Axis_01_Function_Blocks ();
Axis_01_Logic ();
Axis_02_Function_Blocks ();
Axis_02_Logic ();
Axis_03_Function_Blocks ();
Axis_03_Logic ();
Axis_04_Function_Blocks ();
Axis_04_Logic ();
Axis_05_Function_Blocks ();
Axis_05_Logic ();
Axis_06_Function_Blocks ();
Axis_06_Logic ();
Axis_07_Function_Blocks ();
Axis_07_Logic ();
Axis_08_Function_Blocks ();
Axis_08_Logic ();
Axis_09_Function_Blocks ();
Axis_09_Logic ();
Axis_10_Function_Blocks ();
Axis_10_Logic ();
Axis_11_Function_Blocks ();
Axis_11_Logic ();
Axis_12_Function_Blocks ();
Axis_12_Logic ();
Axis_13_Function_Blocks ();
Axis_13_Logic ();
Axis_14_Function_Blocks ();
Axis_14_Logic ();
Axis_15_Function_Blocks ();
Axis_15_Logic ();
Axis_16_Function_Blocks ();
Axis_16_Logic ();
Group_01_Function_Blocks ();
Group_01_Logic ();
Group_02_Function_Blocks ();
Group_02_Logic ();
Group_03_Function_Blocks ();
Group_03_Logic ();
Group_04_Function_Blocks ();
Group_04_Logic ();
Group_05_Function_Blocks ();
Group_05_Logic ();
Group_06_Function_Blocks ();
Group_06_Logic ();
Group_07_Function_Blocks ();
Group_07_Logic ();
Group_08_Function_Blocks ();
Group_08_Logic ();
Indicators ();

END_PROGRAM

// ---- POUs/Axis_01_Function_Blocks.TcPOU
PROGRAM Axis_01_Function_Blocks
VAR
END_VAR

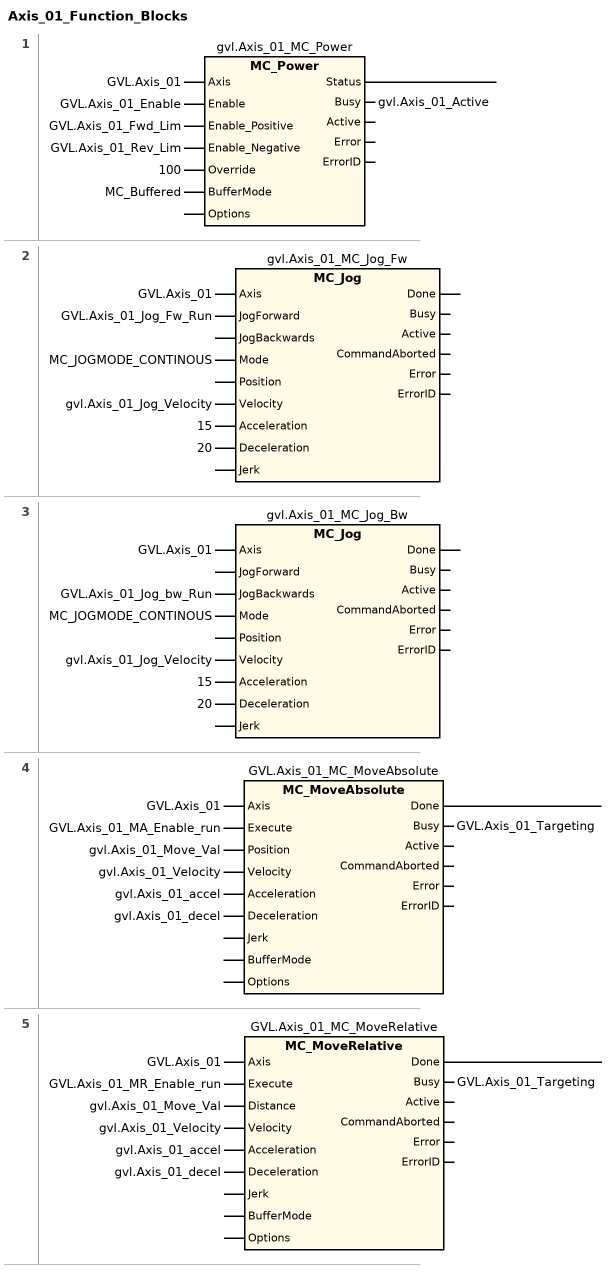
// NETWORK 1
gvl.Axis_01_MC_Power(
    Axis := GVL.Axis_01,
    Enable := GVL.Axis_01_Enable,
    Enable_Positive := GVL.Axis_01_Fwd_Lim,
    Enable_Negative := GVL.Axis_01_Rev_Lim,
    Override := 100,
    BufferMode := MC_Buffered,
    Busy => gvl.Axis_01_Active); // MC_Power

// NETWORK 2
gvl.Axis_01_MC_Jog_Fw(
    Axis := GVL.Axis_01,
    JogForward := GVL.Axis_01_Jog_Fw_Run,
    Mode := MC_JOGMODE_CONTINOUS,
    Velocity := gvl.Axis_01_Jog_Velocity,
    Acceleration := 15,
    Deceleration := 20); // MC_Jog

// NETWORK 3
gvl.Axis_01_MC_Jog_Bw(
    Axis := GVL.Axis_01,
    JogBackwards := GVL.Axis_01_Jog_bw_Run,
    Mode := MC_JOGMODE_CONTINOUS,
    Velocity := gvl.Axis_01_Jog_Velocity,
    Acceleration := 15,
    Deceleration := 20); // MC_Jog

// NETWORK 4
GVL.Axis_01_MC_MoveAbsolute(
    Axis := GVL.Axis_01,
    Execute := GVL.Axis_01_MA_Enable_run,
    Position := gvl.Axis_01_Move_Val,
    Velocity := gvl.Axis_01_Velocity,
    Acceleration := gvl.Axis_01_accel,
    Deceleration := gvl.Axis_01_decel,
    Busy => GVL.Axis_01_Targeting); // MC_MoveAbsolute

// NETWORK 5
GVL.Axis_01_MC_MoveRelative(
    Axis := GVL.Axis_01,
    Execute := GVL.Axis_01_MR_Enable_run,
    Distance := gvl.Axis_01_Move_Val,
    Velocity := gvl.Axis_01_Velocity,
    Acceleration := gvl.Axis_01_accel,
    Deceleration := gvl.Axis_01_decel,
    Busy => GVL.Axis_01_Targeting); // MC_MoveRelative

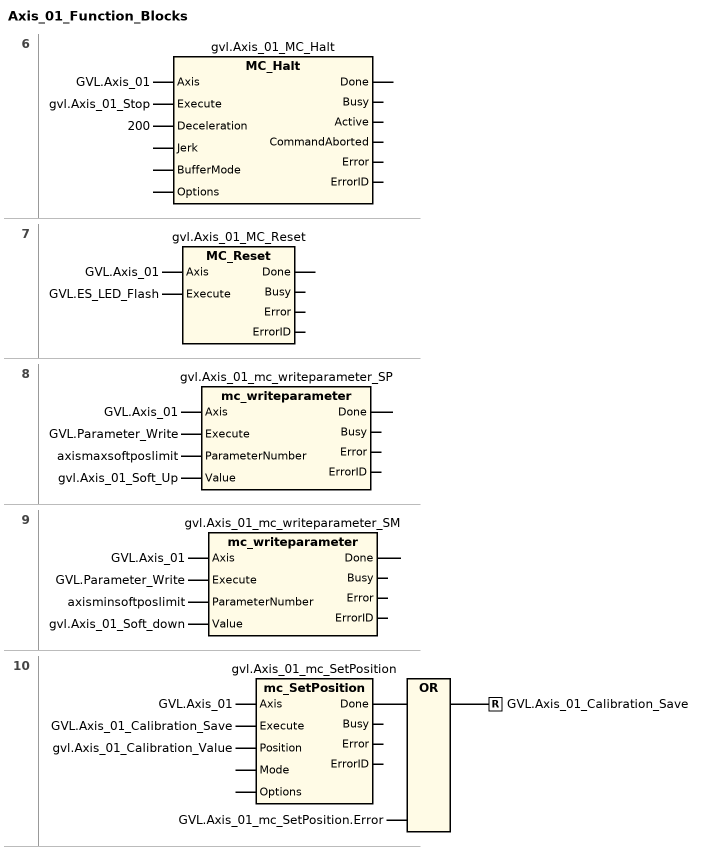
// NETWORK 6
gvl.Axis_01_MC_Halt(Axis := GVL.Axis_01, Execute := gvl.Axis_01_Stop, Deceleration := 200); // MC_Halt

// NETWORK 7
gvl.Axis_01_MC_Reset(Axis := GVL.Axis_01, Execute := GVL.ES_LED_Flash); // MC_Reset

// NETWORK 8
gvl.Axis_01_mc_writeparameter_SP(
    Axis := GVL.Axis_01,
    Execute := GVL.Parameter_Write,
    ParameterNumber := axismaxsoftposlimit,
    Value := gvl.Axis_01_Soft_Up); // mc_writeparameter

// NETWORK 9
gvl.Axis_01_mc_writeparameter_SM(
    Axis := GVL.Axis_01,
    Execute := GVL.Parameter_Write,
    ParameterNumber := axisminsoftposlimit,
    Value := gvl.Axis_01_Soft_down); // mc_writeparameter

// NETWORK 10
gvl.Axis_01_mc_SetPosition(
    Axis := GVL.Axis_01,
    Execute := GVL.Axis_01_Calibration_Save,
    Position := gvl.Axis_01_Calibration_Value); // mc_SetPosition
GVL.Axis_01_Calibration_Save R= gvl.Axis_01_mc_SetPosition.Done OR GVL.Axis_01_mc_SetPosition.Error;

END_PROGRAM

// ---- POUs/Axis_01_Logic.TcPOU
PROGRAM Axis_01_Logic
VAR
	TON_0: TON;
	TON_1: TON;
	TON_2: TON;
	TON_3: TON;
	Axis_01_Velocity_Range: LREAL;
	Axis_01_Velocity_Scale: LREAL;
	Axis_01_Velocity_Raw: LREAL;
	Axis_01_Soft_Range: LREAL;
	Axis_01_Soft_Position: LREAL;
	Axis_01_Soft_Position_In_Range: LREAL;
END_VAR

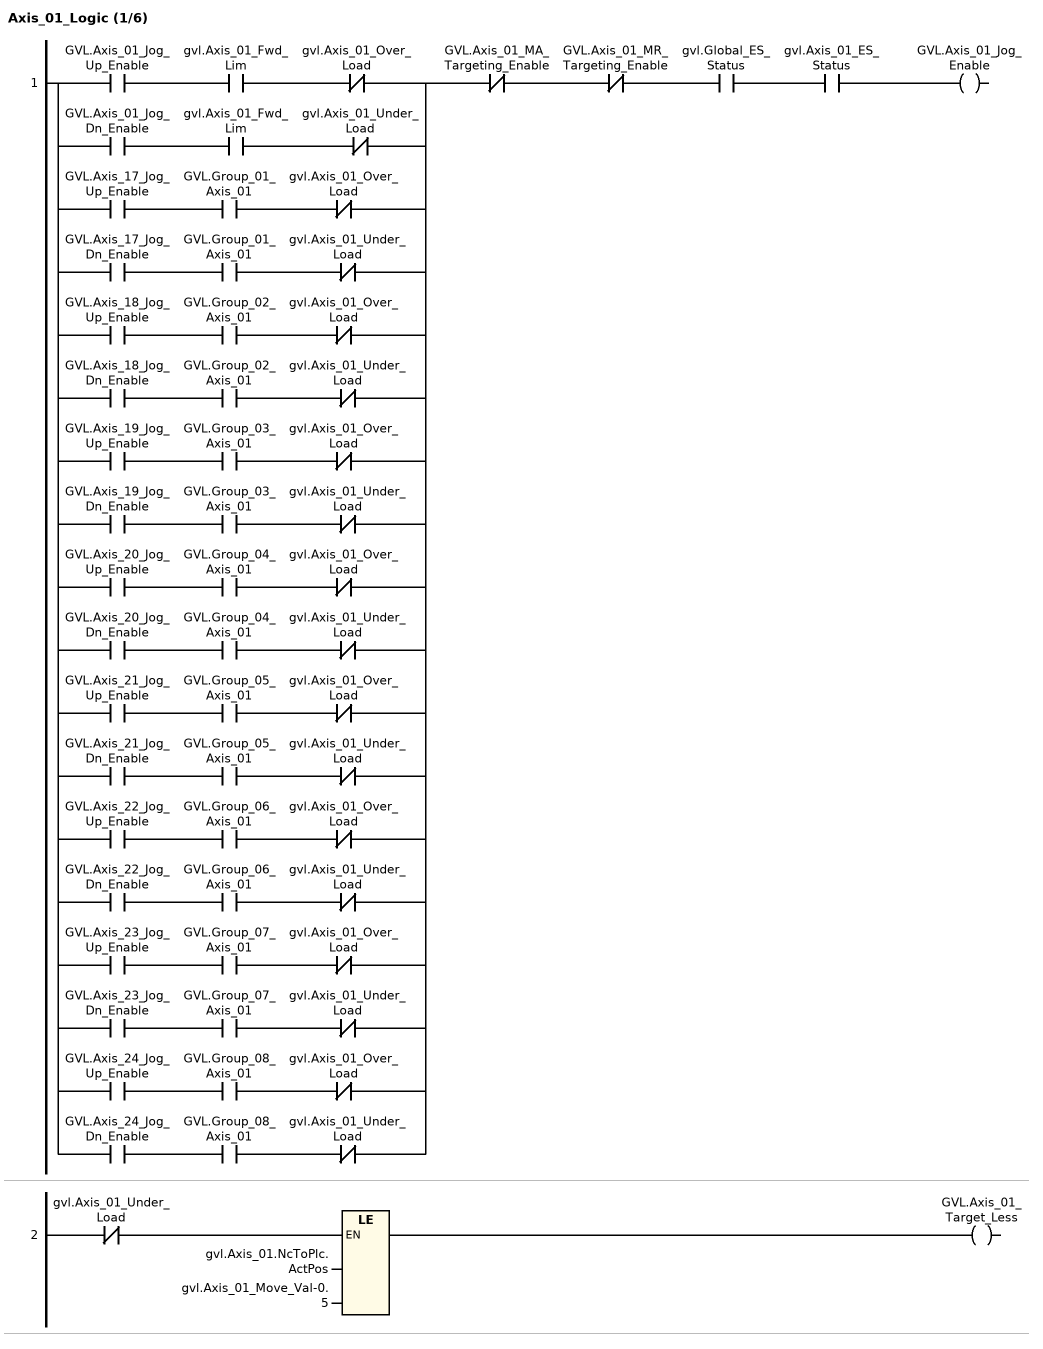
// NETWORK 1
GVL.Axis_01_Jog_Enable := (GVL.Axis_01_Jog_Up_Enable AND gvl.Axis_01_Fwd_Lim AND NOT gvl.Axis_01_Over_Load OR GVL.Axis_01_Jog_Dn_Enable AND gvl.Axis_01_Fwd_Lim AND NOT gvl.Axis_01_Under_Load OR GVL.Axis_17_Jog_Up_Enable AND GVL.Group_01_Axis_01 AND NOT gvl.Axis_01_Over_Load OR GVL.Axis_17_Jog_Dn_Enable AND GVL.Group_01_Axis_01 AND NOT gvl.Axis_01_Under_Load OR GVL.Axis_18_Jog_Up_Enable AND GVL.Group_02_Axis_01 AND NOT gvl.Axis_01_Over_Load OR GVL.Axis_18_Jog_Dn_Enable AND GVL.Group_02_Axis_01 AND NOT gvl.Axis_01_Under_Load OR GVL.Axis_19_Jog_Up_Enable AND GVL.Group_03_Axis_01 AND NOT gvl.Axis_01_Over_Load OR GVL.Axis_19_Jog_Dn_Enable AND GVL.Group_03_Axis_01 AND NOT gvl.Axis_01_Under_Load OR GVL.Axis_20_Jog_Up_Enable AND GVL.Group_04_Axis_01 AND NOT gvl.Axis_01_Over_Load OR GVL.Axis_20_Jog_Dn_Enable AND GVL.Group_04_Axis_01 AND NOT gvl.Axis_01_Under_Load OR GVL.Axis_21_Jog_Up_Enable AND GVL.Group_05_Axis_01 AND NOT gvl.Axis_01_Over_Load OR GVL.Axis_21_Jog_Dn_Enable AND GVL.Group_05_Axis_01 AND NOT gvl.Axis_01_Under_Load OR GVL.Axis_22_Jog_Up_Enable AND GVL.Group_06_Axis_01 AND NOT gvl.Axis_01_Over_Load OR GVL.Axis_22_Jog_Dn_Enable AND GVL.Group_06_Axis_01 AND NOT gvl.Axis_01_Under_Load OR GVL.Axis_23_Jog_Up_Enable AND GVL.Group_07_Axis_01 AND NOT gvl.Axis_01_Over_Load OR GVL.Axis_23_Jog_Dn_Enable AND GVL.Group_07_Axis_01 AND NOT gvl.Axis_01_Under_Load OR GVL.Axis_24_Jog_Up_Enable AND GVL.Group_08_Axis_01 AND NOT gvl.Axis_01_Over_Load OR GVL.Axis_24_Jog_Dn_Enable AND GVL.Group_08_Axis_01 AND NOT gvl.Axis_01_Under_Load) AND NOT GVL.Axis_01_MA_Targeting_Enable AND NOT GVL.Axis_01_MR_Targeting_Enable AND gvl.Global_ES_Status AND gvl.Axis_01_ES_Status;

// NETWORK 2
GVL.Axis_01_Target_Less := NOT gvl.Axis_01_Under_Load AND gvl.Axis_01.NcToPlc.ActPos <= (gvl.Axis_01_Move_Val-0.5);

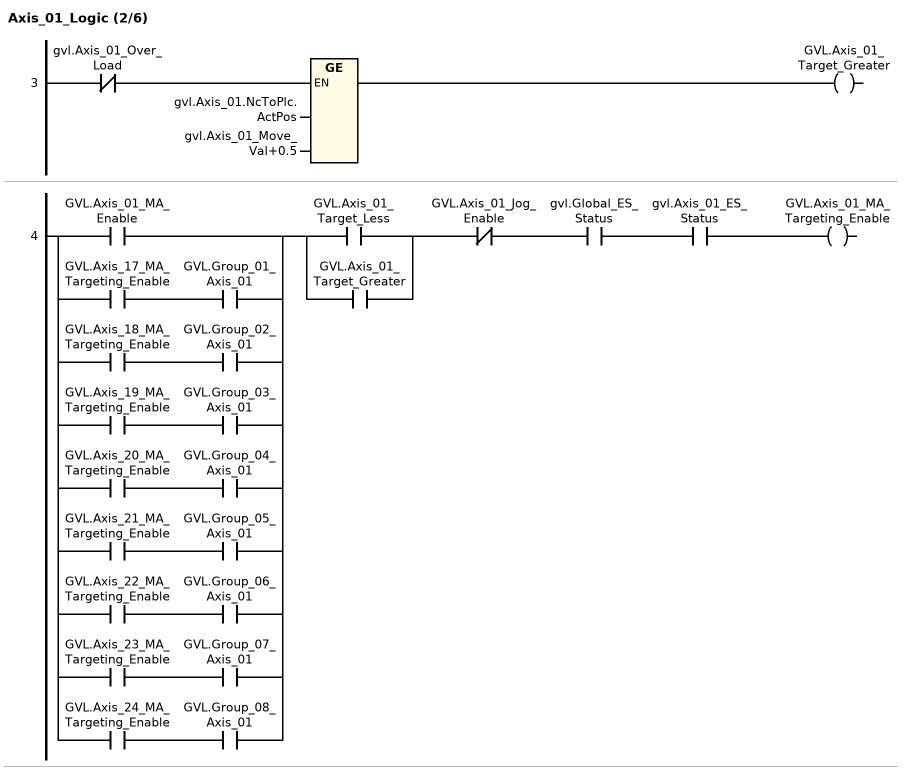
// NETWORK 3
GVL.Axis_01_Target_Greater := NOT gvl.Axis_01_Over_Load AND gvl.Axis_01.NcToPlc.ActPos >= (gvl.Axis_01_Move_Val+0.5);

// NETWORK 4
GVL.Axis_01_MA_Targeting_Enable := (GVL.Axis_01_MA_Enable OR GVL.Axis_17_MA_Targeting_Enable AND GVL.Group_01_Axis_01 OR GVL.Axis_18_MA_Targeting_Enable AND GVL.Group_02_Axis_01 OR GVL.Axis_19_MA_Targeting_Enable AND GVL.Group_03_Axis_01 OR GVL.Axis_20_MA_Targeting_Enable AND GVL.Group_04_Axis_01 OR GVL.Axis_21_MA_Targeting_Enable AND GVL.Group_05_Axis_01 OR GVL.Axis_22_MA_Targeting_Enable AND GVL.Group_06_Axis_01 OR GVL.Axis_23_MA_Targeting_Enable AND GVL.Group_07_Axis_01 OR GVL.Axis_24_MA_Targeting_Enable AND GVL.Group_08_Axis_01) AND (GVL.Axis_01_Target_Less OR GVL.Axis_01_Target_Greater) AND NOT GVL.Axis_01_Jog_Enable AND gvl.Global_ES_Status AND gvl.Axis_01_ES_Status;

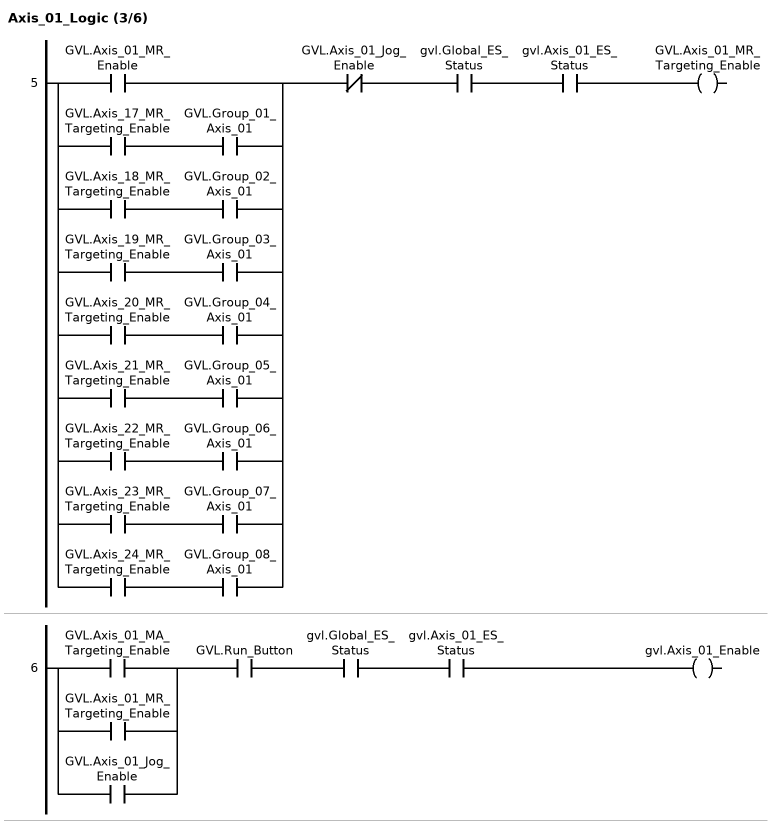
// NETWORK 5
GVL.Axis_01_MR_Targeting_Enable := (GVL.Axis_01_MR_Enable OR GVL.Axis_17_MR_Targeting_Enable AND GVL.Group_01_Axis_01 OR GVL.Axis_18_MR_Targeting_Enable AND GVL.Group_02_Axis_01 OR GVL.Axis_19_MR_Targeting_Enable AND GVL.Group_03_Axis_01 OR GVL.Axis_20_MR_Targeting_Enable AND GVL.Group_04_Axis_01 OR GVL.Axis_21_MR_Targeting_Enable AND GVL.Group_05_Axis_01 OR GVL.Axis_22_MR_Targeting_Enable AND GVL.Group_06_Axis_01 OR GVL.Axis_23_MR_Targeting_Enable AND GVL.Group_07_Axis_01 OR GVL.Axis_24_MR_Targeting_Enable AND GVL.Group_08_Axis_01) AND NOT GVL.Axis_01_Jog_Enable AND gvl.Global_ES_Status AND gvl.Axis_01_ES_Status;

// NETWORK 6
gvl.Axis_01_Enable := (GVL.Axis_01_MA_Targeting_Enable OR GVL.Axis_01_MR_Targeting_Enable OR GVL.Axis_01_Jog_Enable) AND GVL.Run_Button AND gvl.Global_ES_Status AND gvl.Axis_01_ES_Status;

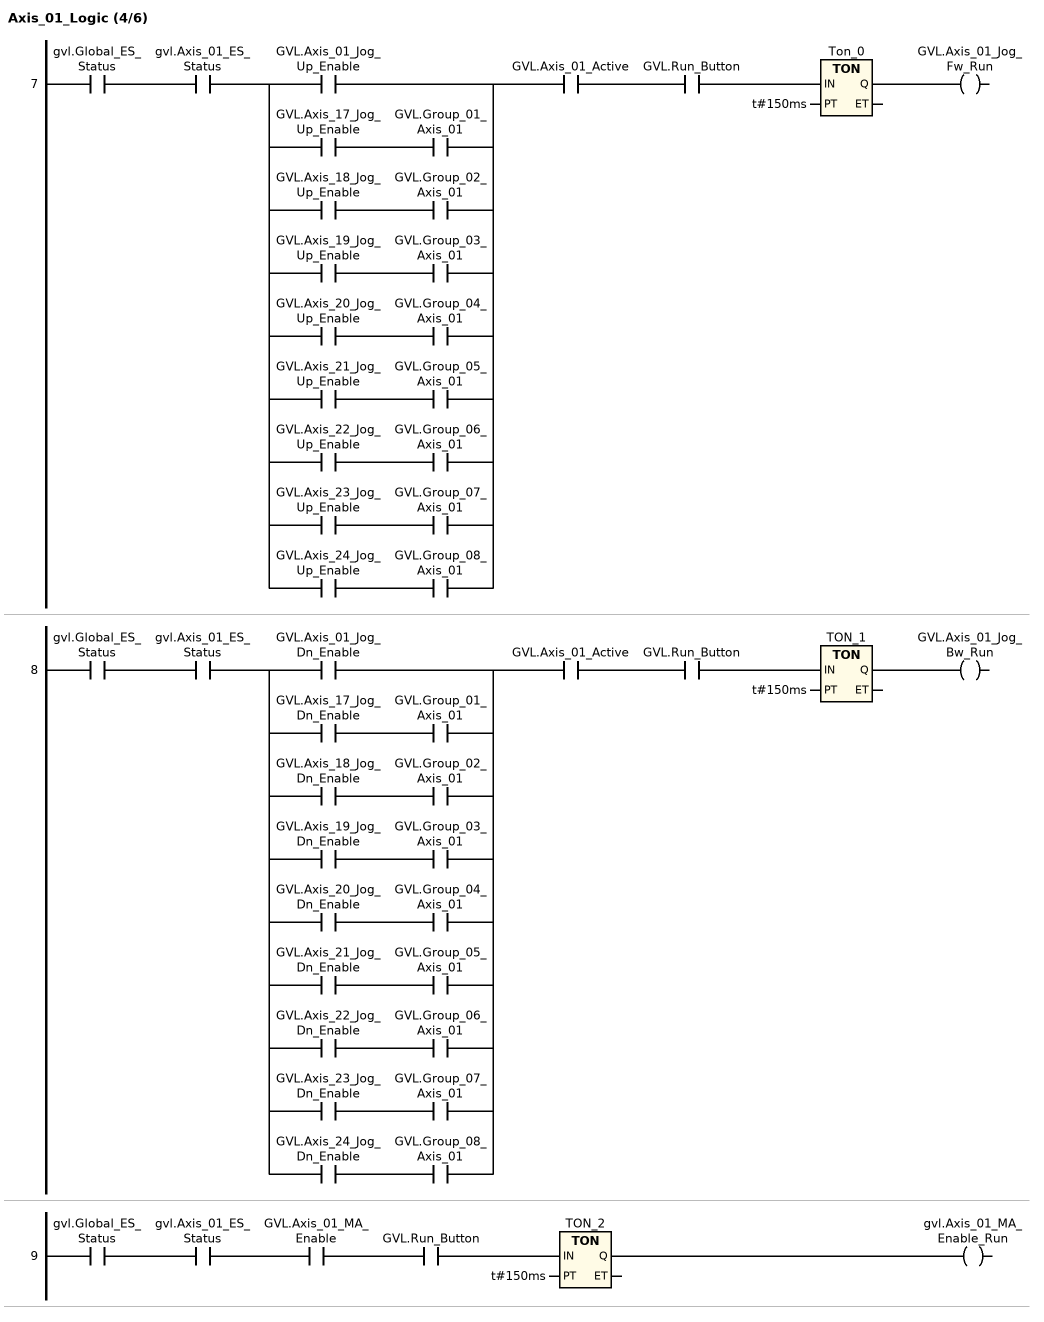
// NETWORK 7
Ton_0(IN := gvl.Global_ES_Status AND gvl.Axis_01_ES_Status AND (GVL.Axis_01_Jog_Up_Enable OR GVL.Axis_17_Jog_Up_Enable AND GVL.Group_01_Axis_01 OR GVL.Axis_18_Jog_Up_Enable AND GVL.Group_02_Axis_01 OR GVL.Axis_19_Jog_Up_Enable AND GVL.Group_03_Axis_01 OR GVL.Axis_20_Jog_Up_Enable AND GVL.Group_04_Axis_01 OR GVL.Axis_21_Jog_Up_Enable AND GVL.Group_05_Axis_01 OR GVL.Axis_22_Jog_Up_Enable AND GVL.Group_06_Axis_01 OR GVL.Axis_23_Jog_Up_Enable AND GVL.Group_07_Axis_01 OR GVL.Axis_24_Jog_Up_Enable AND GVL.Group_08_Axis_01) AND GVL.Axis_01_Active AND GVL.Run_Button, PT := t#150ms); // TON
GVL.Axis_01_Jog_Fw_Run := Ton_0.Q;

// NETWORK 8
TON_1(IN := gvl.Global_ES_Status AND gvl.Axis_01_ES_Status AND (GVL.Axis_01_Jog_Dn_Enable OR GVL.Axis_17_Jog_Dn_Enable AND GVL.Group_01_Axis_01 OR GVL.Axis_18_Jog_Dn_Enable AND GVL.Group_02_Axis_01 OR GVL.Axis_19_Jog_Dn_Enable AND GVL.Group_03_Axis_01 OR GVL.Axis_20_Jog_Dn_Enable AND GVL.Group_04_Axis_01 OR GVL.Axis_21_Jog_Dn_Enable AND GVL.Group_05_Axis_01 OR GVL.Axis_22_Jog_Dn_Enable AND GVL.Group_06_Axis_01 OR GVL.Axis_23_Jog_Dn_Enable AND GVL.Group_07_Axis_01 OR GVL.Axis_24_Jog_Dn_Enable AND GVL.Group_08_Axis_01) AND GVL.Axis_01_Active AND GVL.Run_Button, PT := t#150ms); // TON
GVL.Axis_01_Jog_Bw_Run := TON_1.Q;

// NETWORK 9
TON_2(IN := gvl.Global_ES_Status AND gvl.Axis_01_ES_Status AND GVL.Axis_01_MA_Enable AND GVL.Run_Button, PT := t#150ms); // TON
gvl.Axis_01_MA_Enable_Run := TON_2.Q;

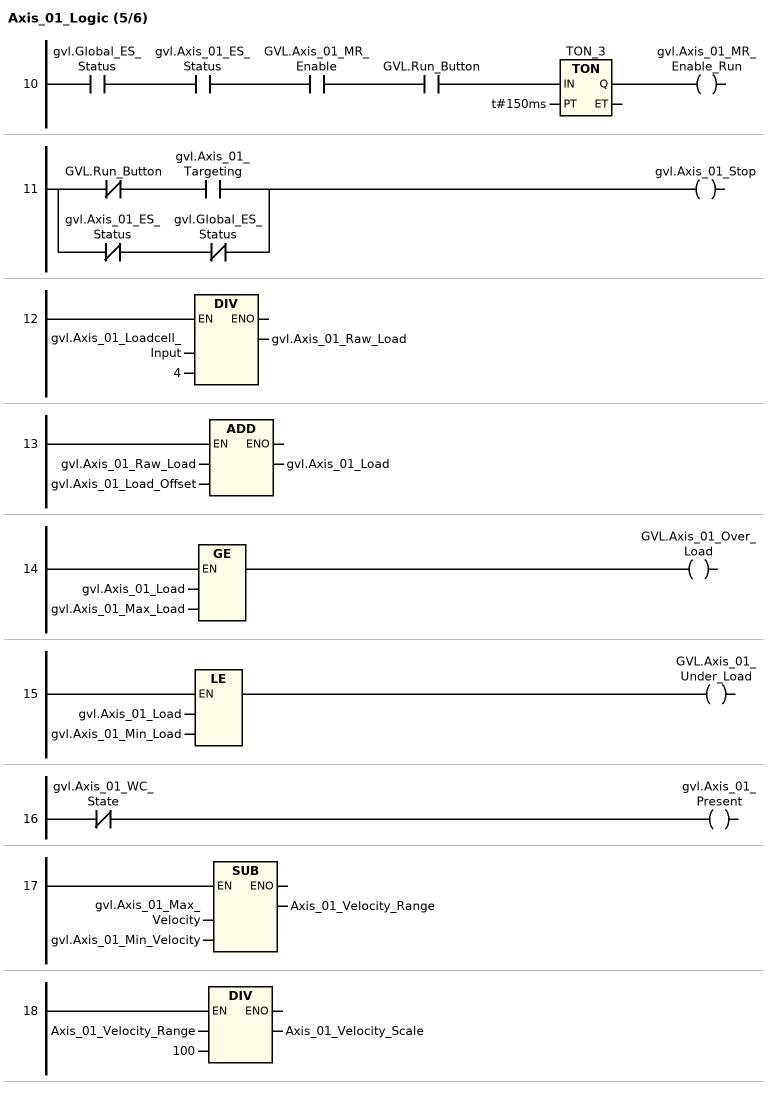
// NETWORK 10
TON_3(IN := gvl.Global_ES_Status AND gvl.Axis_01_ES_Status AND GVL.Axis_01_MR_Enable AND GVL.Run_Button, PT := t#150ms); // TON
gvl.Axis_01_MR_Enable_Run := TON_3.Q;

// NETWORK 11
gvl.Axis_01_Stop := NOT GVL.Run_Button AND gvl.Axis_01_Targeting OR NOT gvl.Axis_01_ES_Status AND NOT gvl.Global_ES_Status;

// NETWORK 12
gvl.Axis_01_Raw_Load := gvl.Axis_01_Loadcell_Input / 4;

// NETWORK 13
gvl.Axis_01_Load := gvl.Axis_01_Raw_Load + gvl.Axis_01_Load_Offset;

// NETWORK 14
GVL.Axis_01_Over_Load := gvl.Axis_01_Load >= gvl.Axis_01_Max_Load;

// NETWORK 15
GVL.Axis_01_Under_Load := gvl.Axis_01_Load <= gvl.Axis_01_Min_Load;

// NETWORK 16
gvl.Axis_01_Present := NOT gvl.Axis_01_WC_State;

// NETWORK 17
Axis_01_Velocity_Range := gvl.Axis_01_Max_Velocity - gvl.Axis_01_Min_Velocity;

// NETWORK 18
Axis_01_Velocity_Scale := Axis_01_Velocity_Range / 100;

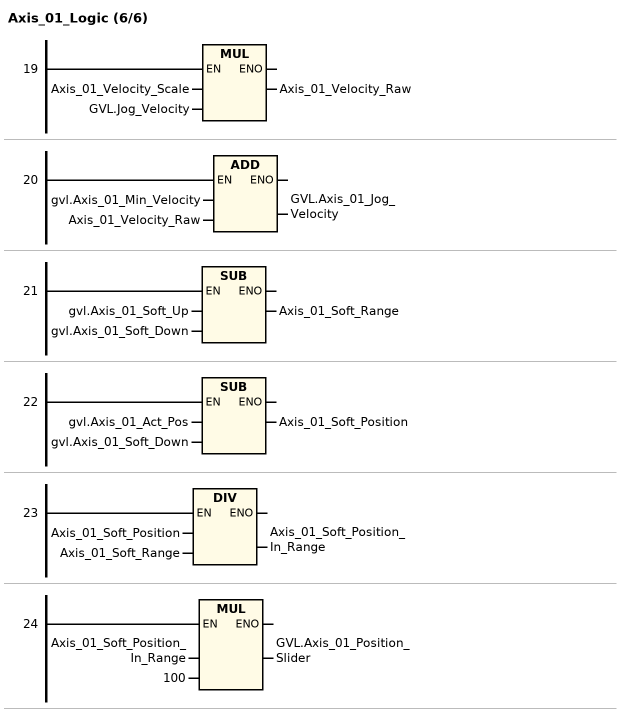
// NETWORK 19
Axis_01_Velocity_Raw := Axis_01_Velocity_Scale * GVL.Jog_Velocity;

// NETWORK 20
GVL.Axis_01_Jog_Velocity := gvl.Axis_01_Min_Velocity + Axis_01_Velocity_Raw;

// NETWORK 21
Axis_01_Soft_Range := gvl.Axis_01_Soft_Up - gvl.Axis_01_Soft_Down;

// NETWORK 22
Axis_01_Soft_Position := gvl.Axis_01_Act_Pos - gvl.Axis_01_Soft_Down;

// NETWORK 23
Axis_01_Soft_Position_In_Range := Axis_01_Soft_Position / Axis_01_Soft_Range;

// NETWORK 24
GVL.Axis_01_Position_Slider := Axis_01_Soft_Position_In_Range * 100;

END_PROGRAM

// ---- POUs/Axis_02_Function_Blocks.TcPOU
PROGRAM Axis_02_Function_Blocks
VAR
END_VAR

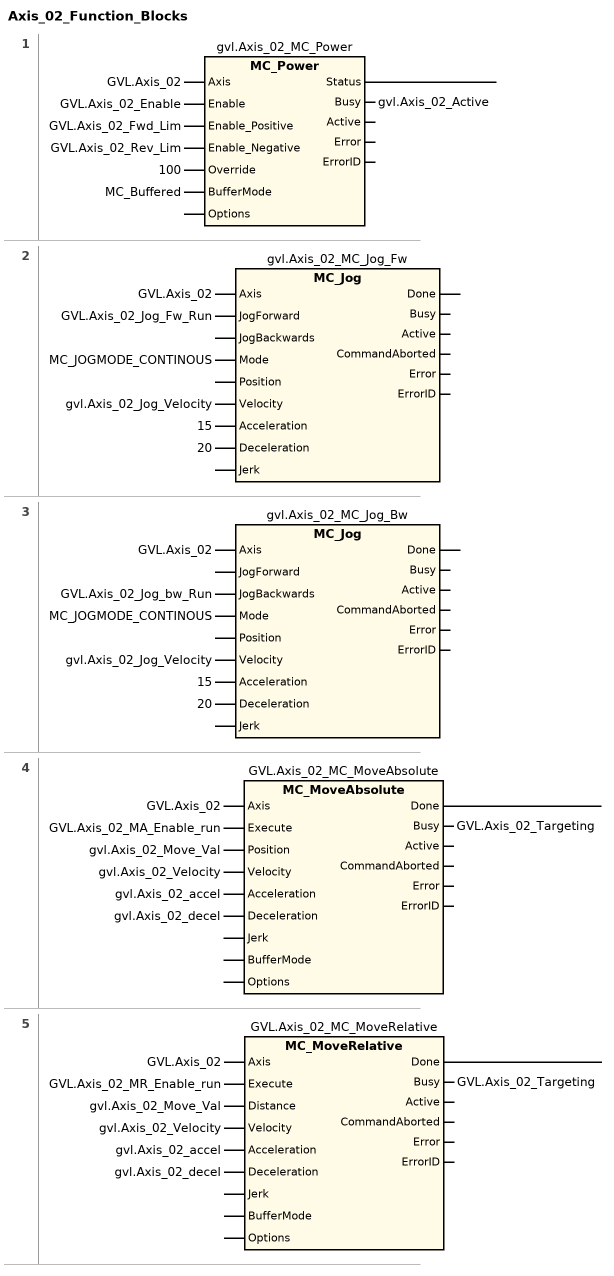
// NETWORK 1
gvl.Axis_02_MC_Power(
    Axis := GVL.Axis_02,
    Enable := GVL.Axis_02_Enable,
    Enable_Positive := GVL.Axis_02_Fwd_Lim,
    Enable_Negative := GVL.Axis_02_Rev_Lim,
    Override := 100,
    BufferMode := MC_Buffered,
    Busy => gvl.Axis_02_Active); // MC_Power

// NETWORK 2
gvl.Axis_02_MC_Jog_Fw(
    Axis := GVL.Axis_02,
    JogForward := GVL.Axis_02_Jog_Fw_Run,
    Mode := MC_JOGMODE_CONTINOUS,
    Velocity := gvl.Axis_02_Jog_Velocity,
    Acceleration := 15,
    Deceleration := 20); // MC_Jog

// NETWORK 3
gvl.Axis_02_MC_Jog_Bw(
    Axis := GVL.Axis_02,
    JogBackwards := GVL.Axis_02_Jog_bw_Run,
    Mode := MC_JOGMODE_CONTINOUS,
    Velocity := gvl.Axis_02_Jog_Velocity,
    Acceleration := 15,
    Deceleration := 20); // MC_Jog

// NETWORK 4
GVL.Axis_02_MC_MoveAbsolute(
    Axis := GVL.Axis_02,
    Execute := GVL.Axis_02_MA_Enable_run,
    Position := gvl.Axis_02_Move_Val,
    Velocity := gvl.Axis_02_Velocity,
    Acceleration := gvl.Axis_02_accel,
    Deceleration := gvl.Axis_02_decel,
    Busy => GVL.Axis_02_Targeting); // MC_MoveAbsolute

// NETWORK 5
GVL.Axis_02_MC_MoveRelative(
    Axis := GVL.Axis_02,
    Execute := GVL.Axis_02_MR_Enable_run,
    Distance := gvl.Axis_02_Move_Val,
    Velocity := gvl.Axis_02_Velocity,
    Acceleration := gvl.Axis_02_accel,
    Deceleration := gvl.Axis_02_decel,
    Busy => GVL.Axis_02_Targeting); // MC_MoveRelative

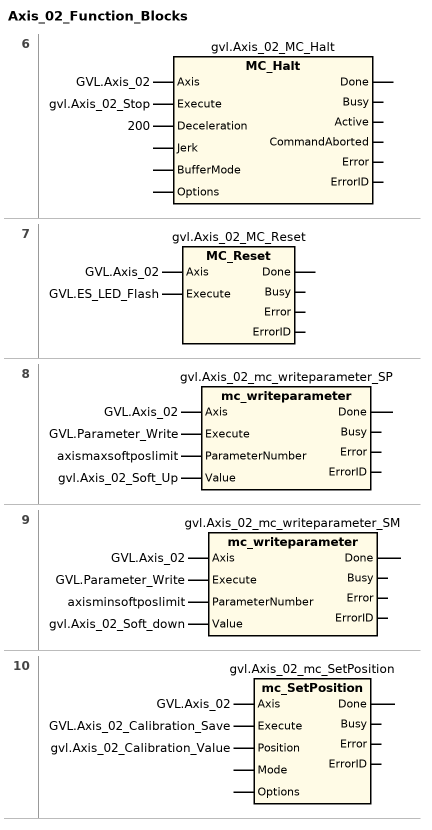
// NETWORK 6
gvl.Axis_02_MC_Halt(Axis := GVL.Axis_02, Execute := gvl.Axis_02_Stop, Deceleration := 200); // MC_Halt

// NETWORK 7
gvl.Axis_02_MC_Reset(Axis := GVL.Axis_02, Execute := GVL.ES_LED_Flash); // MC_Reset

// NETWORK 8
gvl.Axis_02_mc_writeparameter_SP(
    Axis := GVL.Axis_02,
    Execute := GVL.Parameter_Write,
    ParameterNumber := axismaxsoftposlimit,
    Value := gvl.Axis_02_Soft_Up); // mc_writeparameter

// NETWORK 9
gvl.Axis_02_mc_writeparameter_SM(
    Axis := GVL.Axis_02,
    Execute := GVL.Parameter_Write,
    ParameterNumber := axisminsoftposlimit,
    Value := gvl.Axis_02_Soft_down); // mc_writeparameter

// NETWORK 10
gvl.Axis_02_mc_SetPosition(
    Axis := GVL.Axis_02,
    Execute := GVL.Axis_02_Calibration_Save,
    Position := gvl.Axis_02_Calibration_Value); // mc_SetPosition

END_PROGRAM

// ---- POUs/Axis_02_Logic.TcPOU
PROGRAM Axis_02_Logic
VAR
	TON_0: TON;
	TON_1: TON;
	TON_2: TON;
	TON_3: TON;
	Axis_02_Velocity_Range: LREAL;
	Axis_02_Velocity_Scale: LREAL;
	Axis_02_Velocity_Raw: LREAL;
	Axis_02_Soft_Range: LREAL;
	Axis_02_Soft_Position: LREAL;
	Axis_02_Soft_Position_In_Range: LREAL;
END_VAR

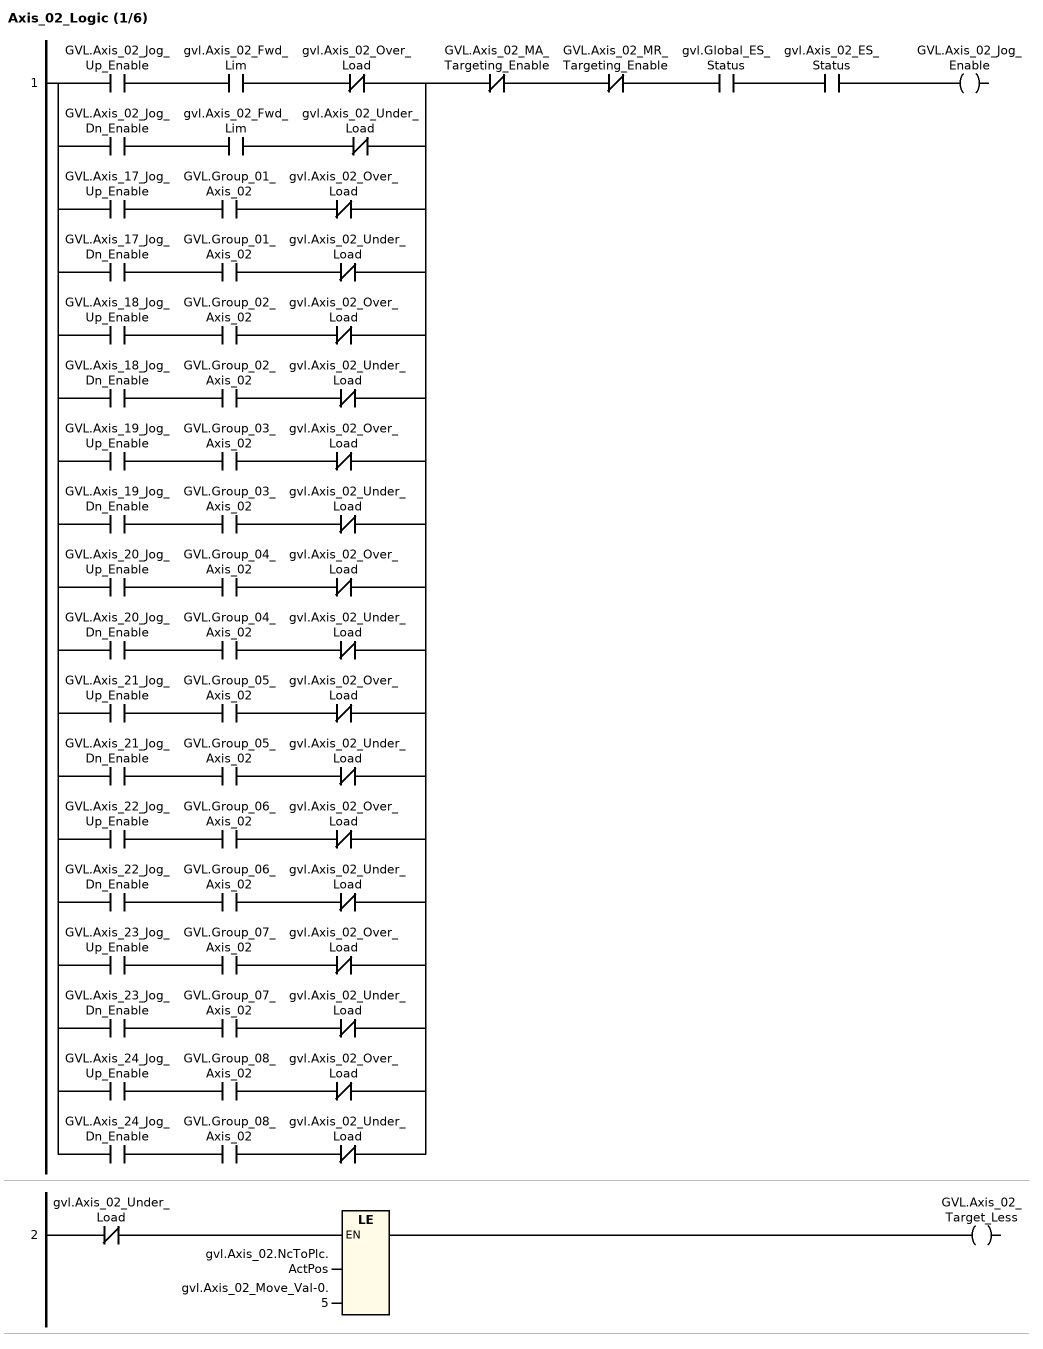
// NETWORK 1
GVL.Axis_02_Jog_Enable := (GVL.Axis_02_Jog_Up_Enable AND gvl.Axis_02_Fwd_Lim AND NOT gvl.Axis_02_Over_Load OR GVL.Axis_02_Jog_Dn_Enable AND gvl.Axis_02_Fwd_Lim AND NOT gvl.Axis_02_Under_Load OR GVL.Axis_17_Jog_Up_Enable AND GVL.Group_01_Axis_02 AND NOT gvl.Axis_02_Over_Load OR GVL.Axis_17_Jog_Dn_Enable AND GVL.Group_01_Axis_02 AND NOT gvl.Axis_02_Under_Load OR GVL.Axis_18_Jog_Up_Enable AND GVL.Group_02_Axis_02 AND NOT gvl.Axis_02_Over_Load OR GVL.Axis_18_Jog_Dn_Enable AND GVL.Group_02_Axis_02 AND NOT gvl.Axis_02_Under_Load OR GVL.Axis_19_Jog_Up_Enable AND GVL.Group_03_Axis_02 AND NOT gvl.Axis_02_Over_Load OR GVL.Axis_19_Jog_Dn_Enable AND GVL.Group_03_Axis_02 AND NOT gvl.Axis_02_Under_Load OR GVL.Axis_20_Jog_Up_Enable AND GVL.Group_04_Axis_02 AND NOT gvl.Axis_02_Over_Load OR GVL.Axis_20_Jog_Dn_Enable AND GVL.Group_04_Axis_02 AND NOT gvl.Axis_02_Under_Load OR GVL.Axis_21_Jog_Up_Enable AND GVL.Group_05_Axis_02 AND NOT gvl.Axis_02_Over_Load OR GVL.Axis_21_Jog_Dn_Enable AND GVL.Group_05_Axis_02 AND NOT gvl.Axis_02_Under_Load OR GVL.Axis_22_Jog_Up_Enable AND GVL.Group_06_Axis_02 AND NOT gvl.Axis_02_Over_Load OR GVL.Axis_22_Jog_Dn_Enable AND GVL.Group_06_Axis_02 AND NOT gvl.Axis_02_Under_Load OR GVL.Axis_23_Jog_Up_Enable AND GVL.Group_07_Axis_02 AND NOT gvl.Axis_02_Over_Load OR GVL.Axis_23_Jog_Dn_Enable AND GVL.Group_07_Axis_02 AND NOT gvl.Axis_02_Under_Load OR GVL.Axis_24_Jog_Up_Enable AND GVL.Group_08_Axis_02 AND NOT gvl.Axis_02_Over_Load OR GVL.Axis_24_Jog_Dn_Enable AND GVL.Group_08_Axis_02 AND NOT gvl.Axis_02_Under_Load) AND NOT GVL.Axis_02_MA_Targeting_Enable AND NOT GVL.Axis_02_MR_Targeting_Enable AND gvl.Global_ES_Status AND gvl.Axis_02_ES_Status;

// NETWORK 2
GVL.Axis_02_Target_Less := NOT gvl.Axis_02_Under_Load AND gvl.Axis_02.NcToPlc.ActPos <= (gvl.Axis_02_Move_Val-0.5);

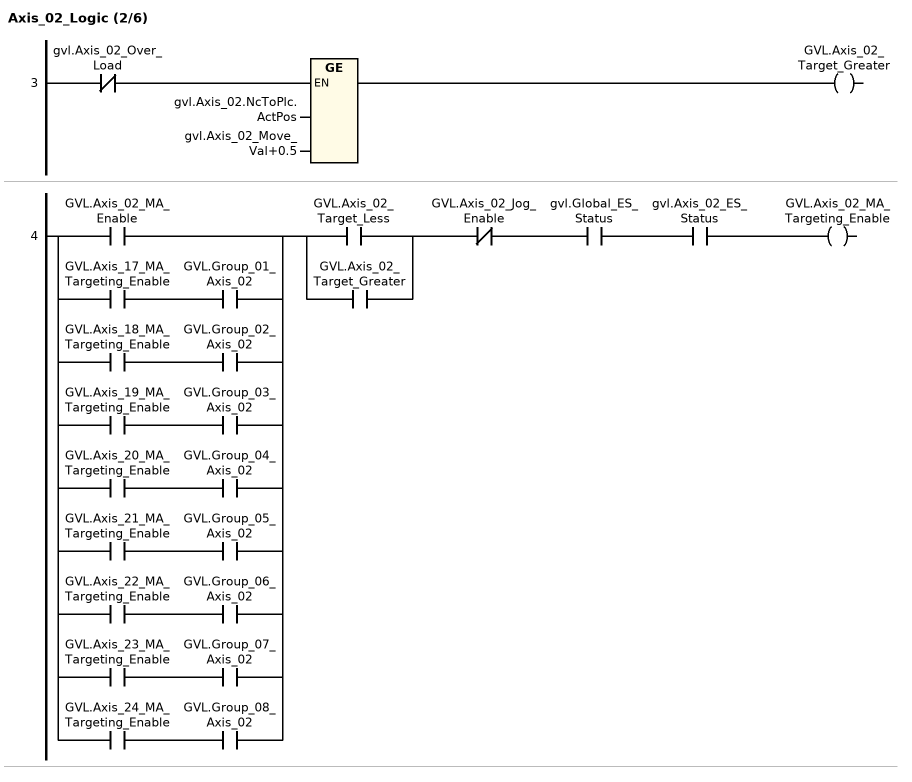
// NETWORK 3
GVL.Axis_02_Target_Greater := NOT gvl.Axis_02_Over_Load AND gvl.Axis_02.NcToPlc.ActPos >= (gvl.Axis_02_Move_Val+0.5);

// NETWORK 4
GVL.Axis_02_MA_Targeting_Enable := (GVL.Axis_02_MA_Enable OR GVL.Axis_17_MA_Targeting_Enable AND GVL.Group_01_Axis_02 OR GVL.Axis_18_MA_Targeting_Enable AND GVL.Group_02_Axis_02 OR GVL.Axis_19_MA_Targeting_Enable AND GVL.Group_03_Axis_02 OR GVL.Axis_20_MA_Targeting_Enable AND GVL.Group_04_Axis_02 OR GVL.Axis_21_MA_Targeting_Enable AND GVL.Group_05_Axis_02 OR GVL.Axis_22_MA_Targeting_Enable AND GVL.Group_06_Axis_02 OR GVL.Axis_23_MA_Targeting_Enable AND GVL.Group_07_Axis_02 OR GVL.Axis_24_MA_Targeting_Enable AND GVL.Group_08_Axis_02) AND (GVL.Axis_02_Target_Less OR GVL.Axis_02_Target_Greater) AND NOT GVL.Axis_02_Jog_Enable AND gvl.Global_ES_Status AND gvl.Axis_02_ES_Status;

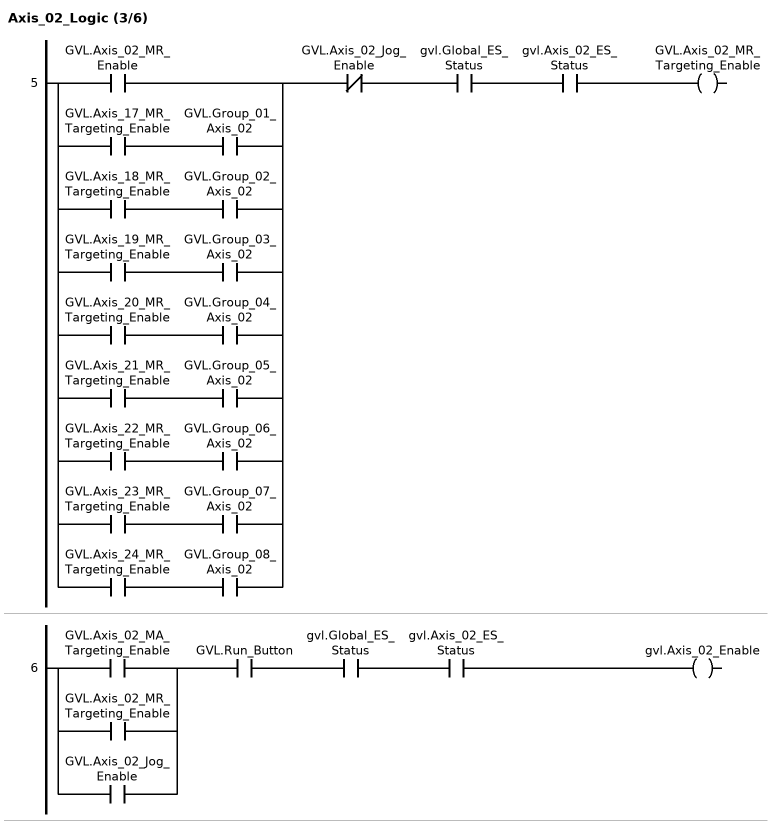
// NETWORK 5
GVL.Axis_02_MR_Targeting_Enable := (GVL.Axis_02_MR_Enable OR GVL.Axis_17_MR_Targeting_Enable AND GVL.Group_01_Axis_02 OR GVL.Axis_18_MR_Targeting_Enable AND GVL.Group_02_Axis_02 OR GVL.Axis_19_MR_Targeting_Enable AND GVL.Group_03_Axis_02 OR GVL.Axis_20_MR_Targeting_Enable AND GVL.Group_04_Axis_02 OR GVL.Axis_21_MR_Targeting_Enable AND GVL.Group_05_Axis_02 OR GVL.Axis_22_MR_Targeting_Enable AND GVL.Group_06_Axis_02 OR GVL.Axis_23_MR_Targeting_Enable AND GVL.Group_07_Axis_02 OR GVL.Axis_24_MR_Targeting_Enable AND GVL.Group_08_Axis_02) AND NOT GVL.Axis_02_Jog_Enable AND gvl.Global_ES_Status AND gvl.Axis_02_ES_Status;

// NETWORK 6
gvl.Axis_02_Enable := (GVL.Axis_02_MA_Targeting_Enable OR GVL.Axis_02_MR_Targeting_Enable OR GVL.Axis_02_Jog_Enable) AND GVL.Run_Button AND gvl.Global_ES_Status AND gvl.Axis_02_ES_Status;

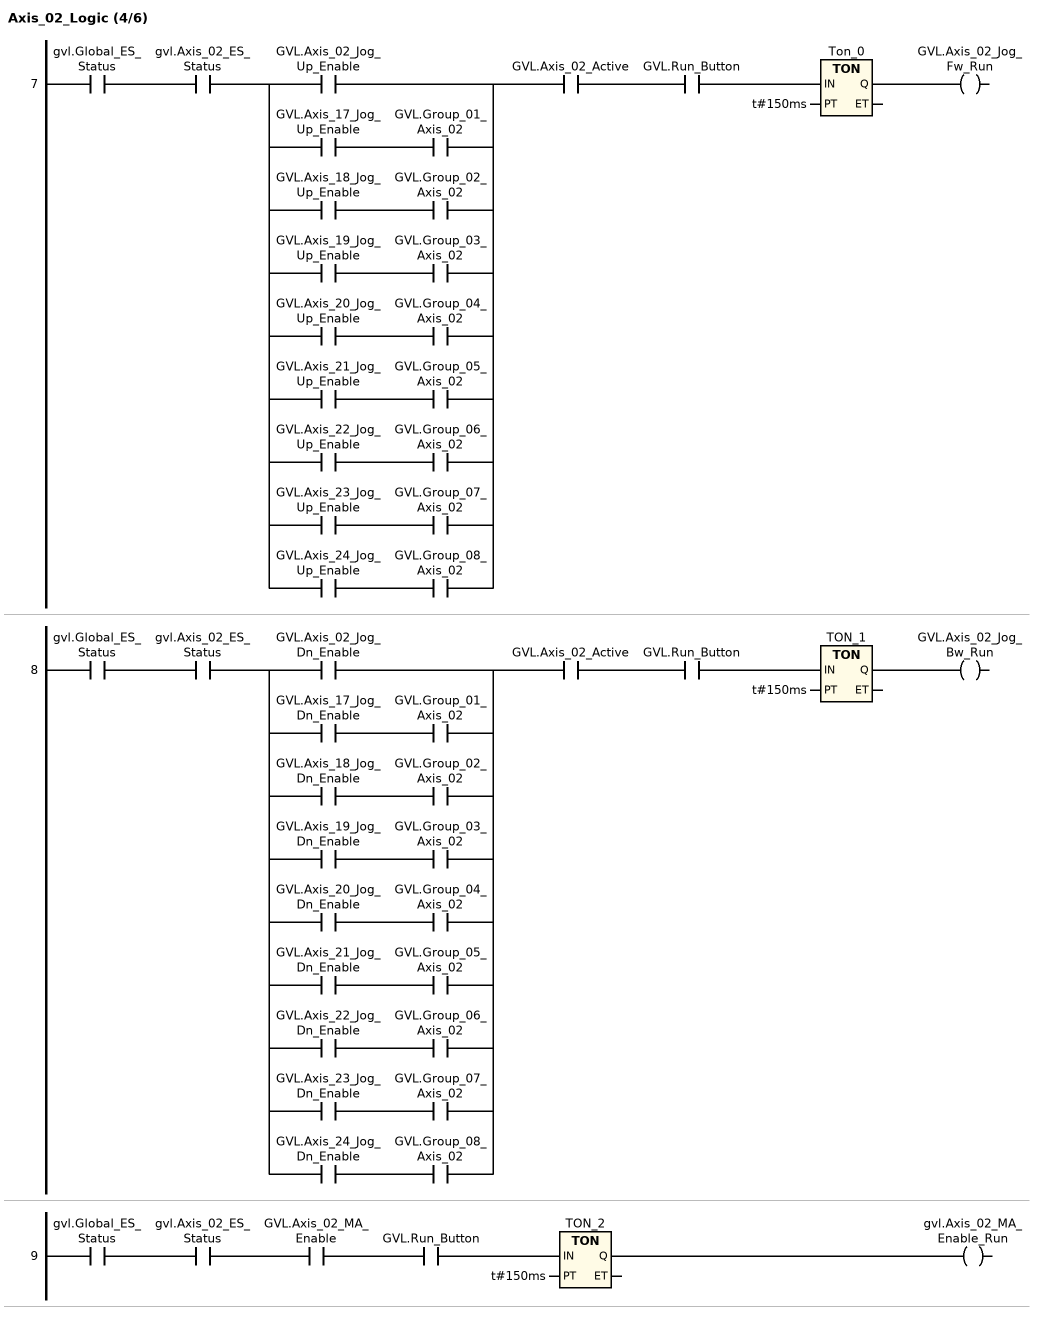
// NETWORK 7
Ton_0(IN := gvl.Global_ES_Status AND gvl.Axis_02_ES_Status AND (GVL.Axis_02_Jog_Up_Enable OR GVL.Axis_17_Jog_Up_Enable AND GVL.Group_01_Axis_02 OR GVL.Axis_18_Jog_Up_Enable AND GVL.Group_02_Axis_02 OR GVL.Axis_19_Jog_Up_Enable AND GVL.Group_03_Axis_02 OR GVL.Axis_20_Jog_Up_Enable AND GVL.Group_04_Axis_02 OR GVL.Axis_21_Jog_Up_Enable AND GVL.Group_05_Axis_02 OR GVL.Axis_22_Jog_Up_Enable AND GVL.Group_06_Axis_02 OR GVL.Axis_23_Jog_Up_Enable AND GVL.Group_07_Axis_02 OR GVL.Axis_24_Jog_Up_Enable AND GVL.Group_08_Axis_02) AND GVL.Axis_02_Active AND GVL.Run_Button, PT := t#150ms); // TON
GVL.Axis_02_Jog_Fw_Run := Ton_0.Q;

// NETWORK 8
TON_1(IN := gvl.Global_ES_Status AND gvl.Axis_02_ES_Status AND (GVL.Axis_02_Jog_Dn_Enable OR GVL.Axis_17_Jog_Dn_Enable AND GVL.Group_01_Axis_02 OR GVL.Axis_18_Jog_Dn_Enable AND GVL.Group_02_Axis_02 OR GVL.Axis_19_Jog_Dn_Enable AND GVL.Group_03_Axis_02 OR GVL.Axis_20_Jog_Dn_Enable AND GVL.Group_04_Axis_02 OR GVL.Axis_21_Jog_Dn_Enable AND GVL.Group_05_Axis_02 OR GVL.Axis_22_Jog_Dn_Enable AND GVL.Group_06_Axis_02 OR GVL.Axis_23_Jog_Dn_Enable AND GVL.Group_07_Axis_02 OR GVL.Axis_24_Jog_Dn_Enable AND GVL.Group_08_Axis_02) AND GVL.Axis_02_Active AND GVL.Run_Button, PT := t#150ms); // TON
GVL.Axis_02_Jog_Bw_Run := TON_1.Q;

// NETWORK 9
TON_2(IN := gvl.Global_ES_Status AND gvl.Axis_02_ES_Status AND GVL.Axis_02_MA_Enable AND GVL.Run_Button, PT := t#150ms); // TON
gvl.Axis_02_MA_Enable_Run := TON_2.Q;

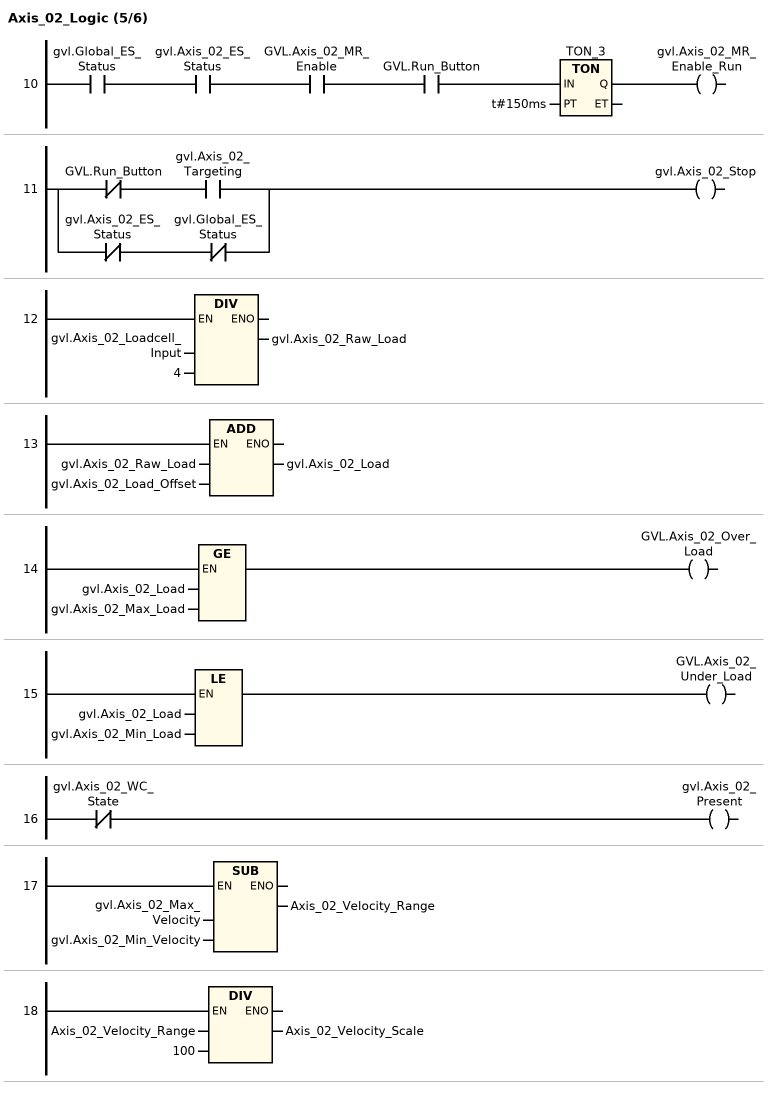
// NETWORK 10
TON_3(IN := gvl.Global_ES_Status AND gvl.Axis_02_ES_Status AND GVL.Axis_02_MR_Enable AND GVL.Run_Button, PT := t#150ms); // TON
gvl.Axis_02_MR_Enable_Run := TON_3.Q;

// NETWORK 11
gvl.Axis_02_Stop := NOT GVL.Run_Button AND gvl.Axis_02_Targeting OR NOT gvl.Axis_02_ES_Status AND NOT gvl.Global_ES_Status;

// NETWORK 12
gvl.Axis_02_Raw_Load := gvl.Axis_02_Loadcell_Input / 4;

// NETWORK 13
gvl.Axis_02_Load := gvl.Axis_02_Raw_Load + gvl.Axis_02_Load_Offset;

// NETWORK 14
GVL.Axis_02_Over_Load := gvl.Axis_02_Load >= gvl.Axis_02_Max_Load;

// NETWORK 15
GVL.Axis_02_Under_Load := gvl.Axis_02_Load <= gvl.Axis_02_Min_Load;

// NETWORK 16
gvl.Axis_02_Present := NOT gvl.Axis_02_WC_State;

// NETWORK 17
Axis_02_Velocity_Range := gvl.Axis_02_Max_Velocity - gvl.Axis_02_Min_Velocity;

// NETWORK 18
Axis_02_Velocity_Scale := Axis_02_Velocity_Range / 100;

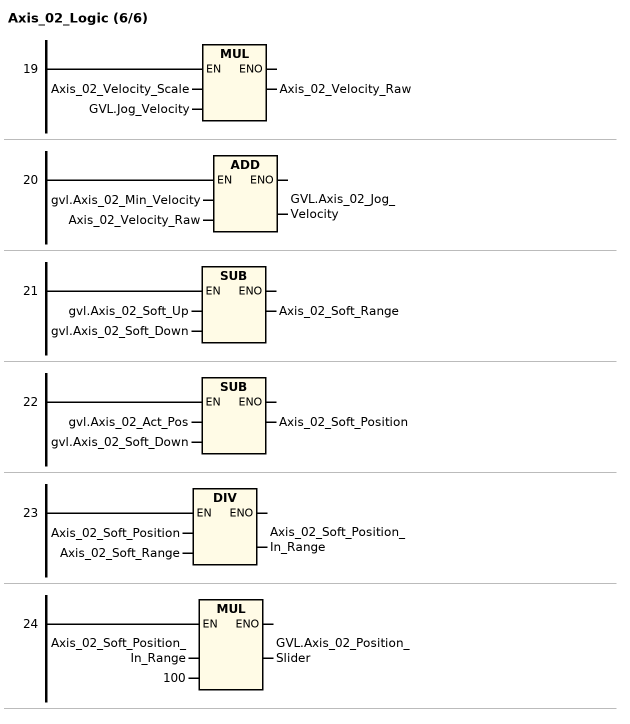
// NETWORK 19
Axis_02_Velocity_Raw := Axis_02_Velocity_Scale * GVL.Jog_Velocity;

// NETWORK 20
GVL.Axis_02_Jog_Velocity := gvl.Axis_02_Min_Velocity + Axis_02_Velocity_Raw;

// NETWORK 21
Axis_02_Soft_Range := gvl.Axis_02_Soft_Up - gvl.Axis_02_Soft_Down;

// NETWORK 22
Axis_02_Soft_Position := gvl.Axis_02_Act_Pos - gvl.Axis_02_Soft_Down;

// NETWORK 23
Axis_02_Soft_Position_In_Range := Axis_02_Soft_Position / Axis_02_Soft_Range;

// NETWORK 24
GVL.Axis_02_Position_Slider := Axis_02_Soft_Position_In_Range * 100;

END_PROGRAM

// ---- POUs/Axis_03_Function_Blocks.TcPOU
PROGRAM Axis_03_Function_Blocks
VAR
END_VAR

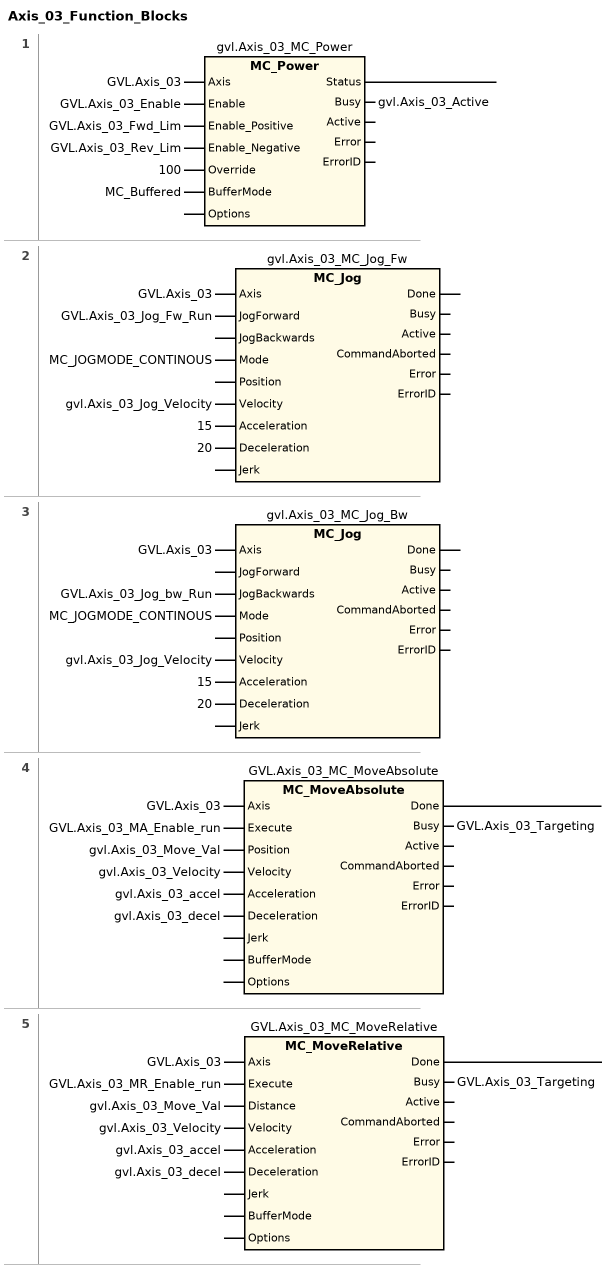
// NETWORK 1
gvl.Axis_03_MC_Power(
    Axis := GVL.Axis_03,
    Enable := GVL.Axis_03_Enable,
    Enable_Positive := GVL.Axis_03_Fwd_Lim,
    Enable_Negative := GVL.Axis_03_Rev_Lim,
    Override := 100,
    BufferMode := MC_Buffered,
    Busy => gvl.Axis_03_Active); // MC_Power

// NETWORK 2
gvl.Axis_03_MC_Jog_Fw(
    Axis := GVL.Axis_03,
    JogForward := GVL.Axis_03_Jog_Fw_Run,
    Mode := MC_JOGMODE_CONTINOUS,
    Velocity := gvl.Axis_03_Jog_Velocity,
    Acceleration := 15,
    Deceleration := 20); // MC_Jog

// NETWORK 3
gvl.Axis_03_MC_Jog_Bw(
    Axis := GVL.Axis_03,
    JogBackwards := GVL.Axis_03_Jog_bw_Run,
    Mode := MC_JOGMODE_CONTINOUS,
    Velocity := gvl.Axis_03_Jog_Velocity,
    Acceleration := 15,
    Deceleration := 20); // MC_Jog

// NETWORK 4
GVL.Axis_03_MC_MoveAbsolute(
    Axis := GVL.Axis_03,
    Execute := GVL.Axis_03_MA_Enable_run,
    Position := gvl.Axis_03_Move_Val,
    Velocity := gvl.Axis_03_Velocity,
    Acceleration := gvl.Axis_03_accel,
    Deceleration := gvl.Axis_03_decel,
    Busy => GVL.Axis_03_Targeting); // MC_MoveAbsolute

// NETWORK 5
GVL.Axis_03_MC_MoveRelative(
    Axis := GVL.Axis_03,
    Execute := GVL.Axis_03_MR_Enable_run,
    Distance := gvl.Axis_03_Move_Val,
    Velocity := gvl.Axis_03_Velocity,
    Acceleration := gvl.Axis_03_accel,
    Deceleration := gvl.Axis_03_decel,
    Busy => GVL.Axis_03_Targeting); // MC_MoveRelative

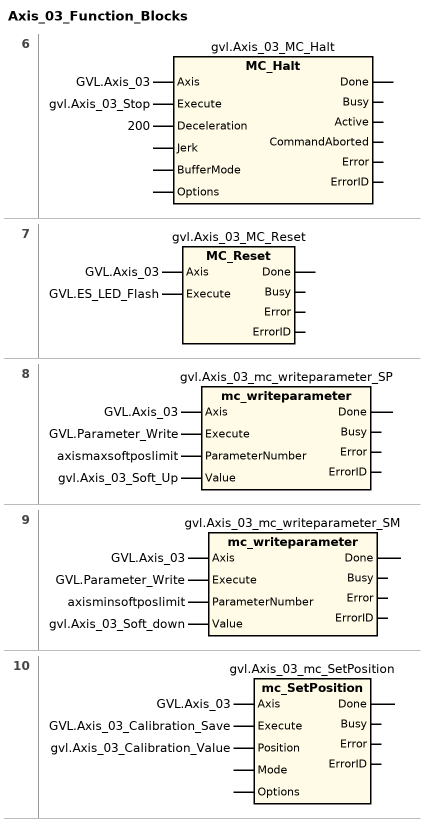
// NETWORK 6
gvl.Axis_03_MC_Halt(Axis := GVL.Axis_03, Execute := gvl.Axis_03_Stop, Deceleration := 200); // MC_Halt

// NETWORK 7
gvl.Axis_03_MC_Reset(Axis := GVL.Axis_03, Execute := GVL.ES_LED_Flash); // MC_Reset

// NETWORK 8
gvl.Axis_03_mc_writeparameter_SP(
    Axis := GVL.Axis_03,
    Execute := GVL.Parameter_Write,
    ParameterNumber := axismaxsoftposlimit,
    Value := gvl.Axis_03_Soft_Up); // mc_writeparameter

// NETWORK 9
gvl.Axis_03_mc_writeparameter_SM(
    Axis := GVL.Axis_03,
    Execute := GVL.Parameter_Write,
    ParameterNumber := axisminsoftposlimit,
    Value := gvl.Axis_03_Soft_down); // mc_writeparameter

// NETWORK 10
gvl.Axis_03_mc_SetPosition(
    Axis := GVL.Axis_03,
    Execute := GVL.Axis_03_Calibration_Save,
    Position := gvl.Axis_03_Calibration_Value); // mc_SetPosition

END_PROGRAM

// ---- POUs/Axis_03_Logic.TcPOU
PROGRAM Axis_03_Logic
VAR
	TON_0: TON;
	TON_1: TON;
	TON_2: TON;
	TON_3: TON;
	Axis_03_Velocity_Range: LREAL;
	Axis_03_Velocity_Scale: LREAL;
	Axis_03_Velocity_Raw: LREAL;
	Axis_03_Soft_Range: LREAL;
	Axis_03_Soft_Position: LREAL;
	Axis_03_Soft_Position_In_Range: LREAL;
END_VAR

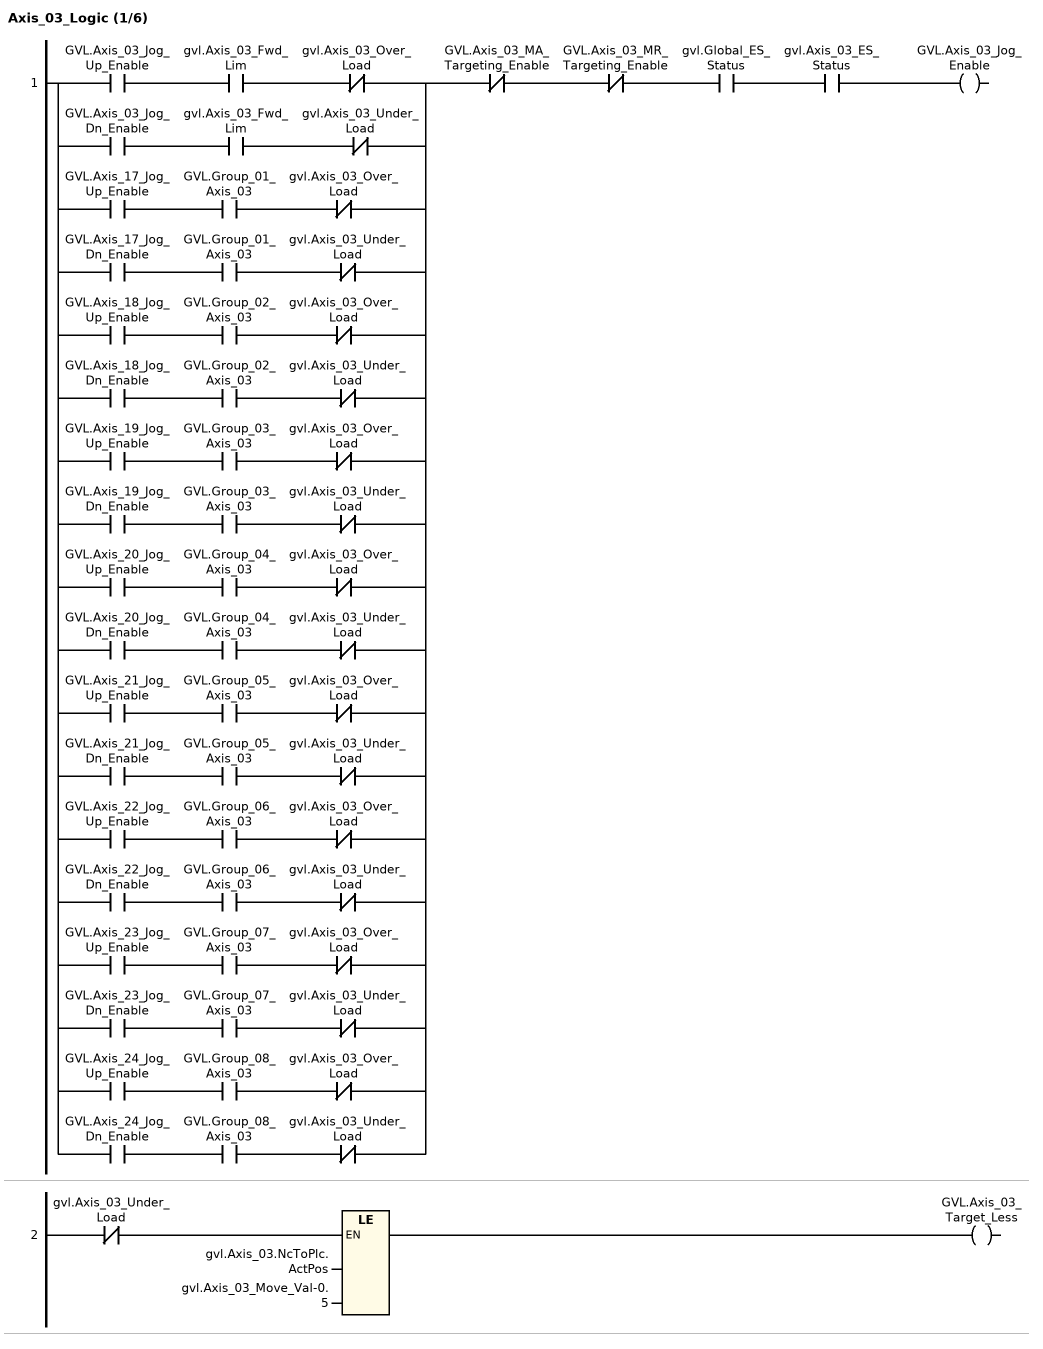
// NETWORK 1
GVL.Axis_03_Jog_Enable := (GVL.Axis_03_Jog_Up_Enable AND gvl.Axis_03_Fwd_Lim AND NOT gvl.Axis_03_Over_Load OR GVL.Axis_03_Jog_Dn_Enable AND gvl.Axis_03_Fwd_Lim AND NOT gvl.Axis_03_Under_Load OR GVL.Axis_17_Jog_Up_Enable AND GVL.Group_01_Axis_03 AND NOT gvl.Axis_03_Over_Load OR GVL.Axis_17_Jog_Dn_Enable AND GVL.Group_01_Axis_03 AND NOT gvl.Axis_03_Under_Load OR GVL.Axis_18_Jog_Up_Enable AND GVL.Group_02_Axis_03 AND NOT gvl.Axis_03_Over_Load OR GVL.Axis_18_Jog_Dn_Enable AND GVL.Group_02_Axis_03 AND NOT gvl.Axis_03_Under_Load OR GVL.Axis_19_Jog_Up_Enable AND GVL.Group_03_Axis_03 AND NOT gvl.Axis_03_Over_Load OR GVL.Axis_19_Jog_Dn_Enable AND GVL.Group_03_Axis_03 AND NOT gvl.Axis_03_Under_Load OR GVL.Axis_20_Jog_Up_Enable AND GVL.Group_04_Axis_03 AND NOT gvl.Axis_03_Over_Load OR GVL.Axis_20_Jog_Dn_Enable AND GVL.Group_04_Axis_03 AND NOT gvl.Axis_03_Under_Load OR GVL.Axis_21_Jog_Up_Enable AND GVL.Group_05_Axis_03 AND NOT gvl.Axis_03_Over_Load OR GVL.Axis_21_Jog_Dn_Enable AND GVL.Group_05_Axis_03 AND NOT gvl.Axis_03_Under_Load OR GVL.Axis_22_Jog_Up_Enable AND GVL.Group_06_Axis_03 AND NOT gvl.Axis_03_Over_Load OR GVL.Axis_22_Jog_Dn_Enable AND GVL.Group_06_Axis_03 AND NOT gvl.Axis_03_Under_Load OR GVL.Axis_23_Jog_Up_Enable AND GVL.Group_07_Axis_03 AND NOT gvl.Axis_03_Over_Load OR GVL.Axis_23_Jog_Dn_Enable AND GVL.Group_07_Axis_03 AND NOT gvl.Axis_03_Under_Load OR GVL.Axis_24_Jog_Up_Enable AND GVL.Group_08_Axis_03 AND NOT gvl.Axis_03_Over_Load OR GVL.Axis_24_Jog_Dn_Enable AND GVL.Group_08_Axis_03 AND NOT gvl.Axis_03_Under_Load) AND NOT GVL.Axis_03_MA_Targeting_Enable AND NOT GVL.Axis_03_MR_Targeting_Enable AND gvl.Global_ES_Status AND gvl.Axis_03_ES_Status;

// NETWORK 2
GVL.Axis_03_Target_Less := NOT gvl.Axis_03_Under_Load AND gvl.Axis_03.NcToPlc.ActPos <= (gvl.Axis_03_Move_Val-0.5);

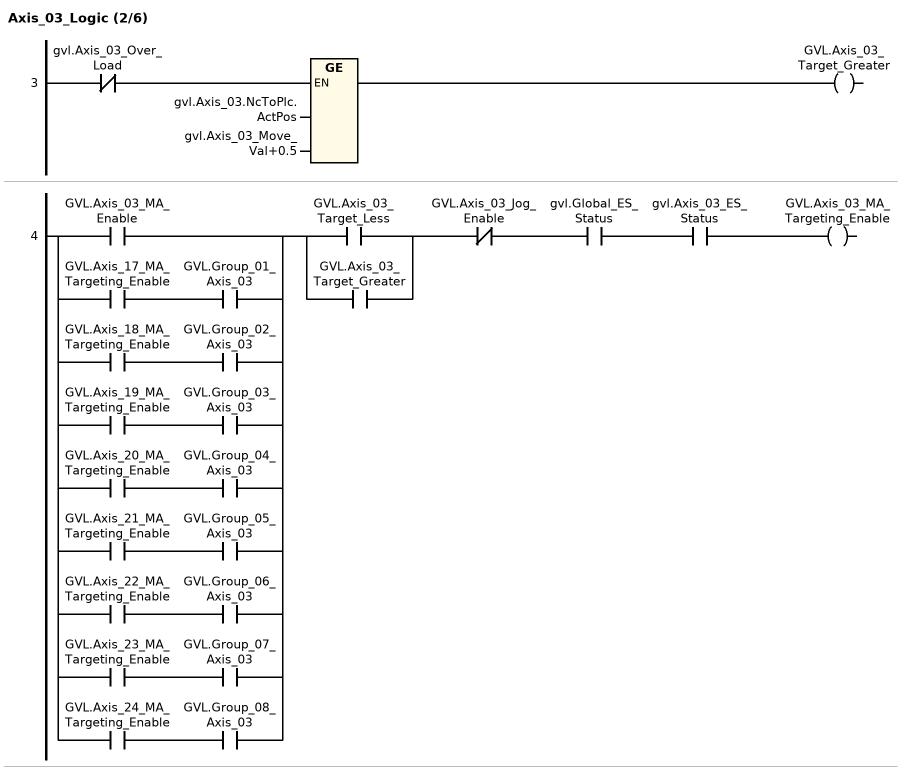
// NETWORK 3
GVL.Axis_03_Target_Greater := NOT gvl.Axis_03_Over_Load AND gvl.Axis_03.NcToPlc.ActPos >= (gvl.Axis_03_Move_Val+0.5);

// NETWORK 4
GVL.Axis_03_MA_Targeting_Enable := (GVL.Axis_03_MA_Enable OR GVL.Axis_17_MA_Targeting_Enable AND GVL.Group_01_Axis_03 OR GVL.Axis_18_MA_Targeting_Enable AND GVL.Group_02_Axis_03 OR GVL.Axis_19_MA_Targeting_Enable AND GVL.Group_03_Axis_03 OR GVL.Axis_20_MA_Targeting_Enable AND GVL.Group_04_Axis_03 OR GVL.Axis_21_MA_Targeting_Enable AND GVL.Group_05_Axis_03 OR GVL.Axis_22_MA_Targeting_Enable AND GVL.Group_06_Axis_03 OR GVL.Axis_23_MA_Targeting_Enable AND GVL.Group_07_Axis_03 OR GVL.Axis_24_MA_Targeting_Enable AND GVL.Group_08_Axis_03) AND (GVL.Axis_03_Target_Less OR GVL.Axis_03_Target_Greater) AND NOT GVL.Axis_03_Jog_Enable AND gvl.Global_ES_Status AND gvl.Axis_03_ES_Status;

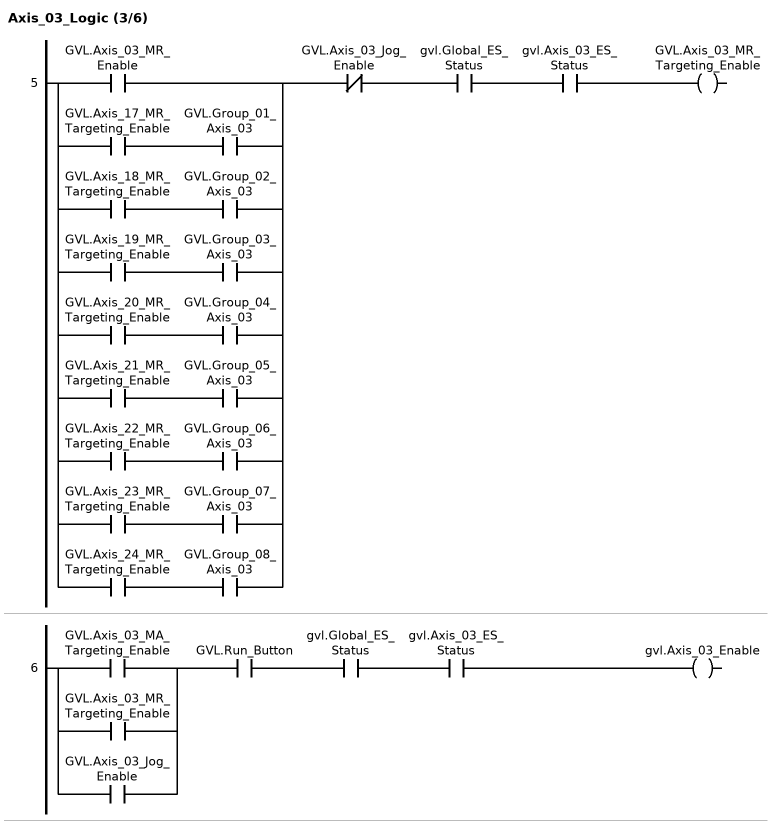
// NETWORK 5
GVL.Axis_03_MR_Targeting_Enable := (GVL.Axis_03_MR_Enable OR GVL.Axis_17_MR_Targeting_Enable AND GVL.Group_01_Axis_03 OR GVL.Axis_18_MR_Targeting_Enable AND GVL.Group_02_Axis_03 OR GVL.Axis_19_MR_Targeting_Enable AND GVL.Group_03_Axis_03 OR GVL.Axis_20_MR_Targeting_Enable AND GVL.Group_04_Axis_03 OR GVL.Axis_21_MR_Targeting_Enable AND GVL.Group_05_Axis_03 OR GVL.Axis_22_MR_Targeting_Enable AND GVL.Group_06_Axis_03 OR GVL.Axis_23_MR_Targeting_Enable AND GVL.Group_07_Axis_03 OR GVL.Axis_24_MR_Targeting_Enable AND GVL.Group_08_Axis_03) AND NOT GVL.Axis_03_Jog_Enable AND gvl.Global_ES_Status AND gvl.Axis_03_ES_Status;

// NETWORK 6
gvl.Axis_03_Enable := (GVL.Axis_03_MA_Targeting_Enable OR GVL.Axis_03_MR_Targeting_Enable OR GVL.Axis_03_Jog_Enable) AND GVL.Run_Button AND gvl.Global_ES_Status AND gvl.Axis_03_ES_Status;

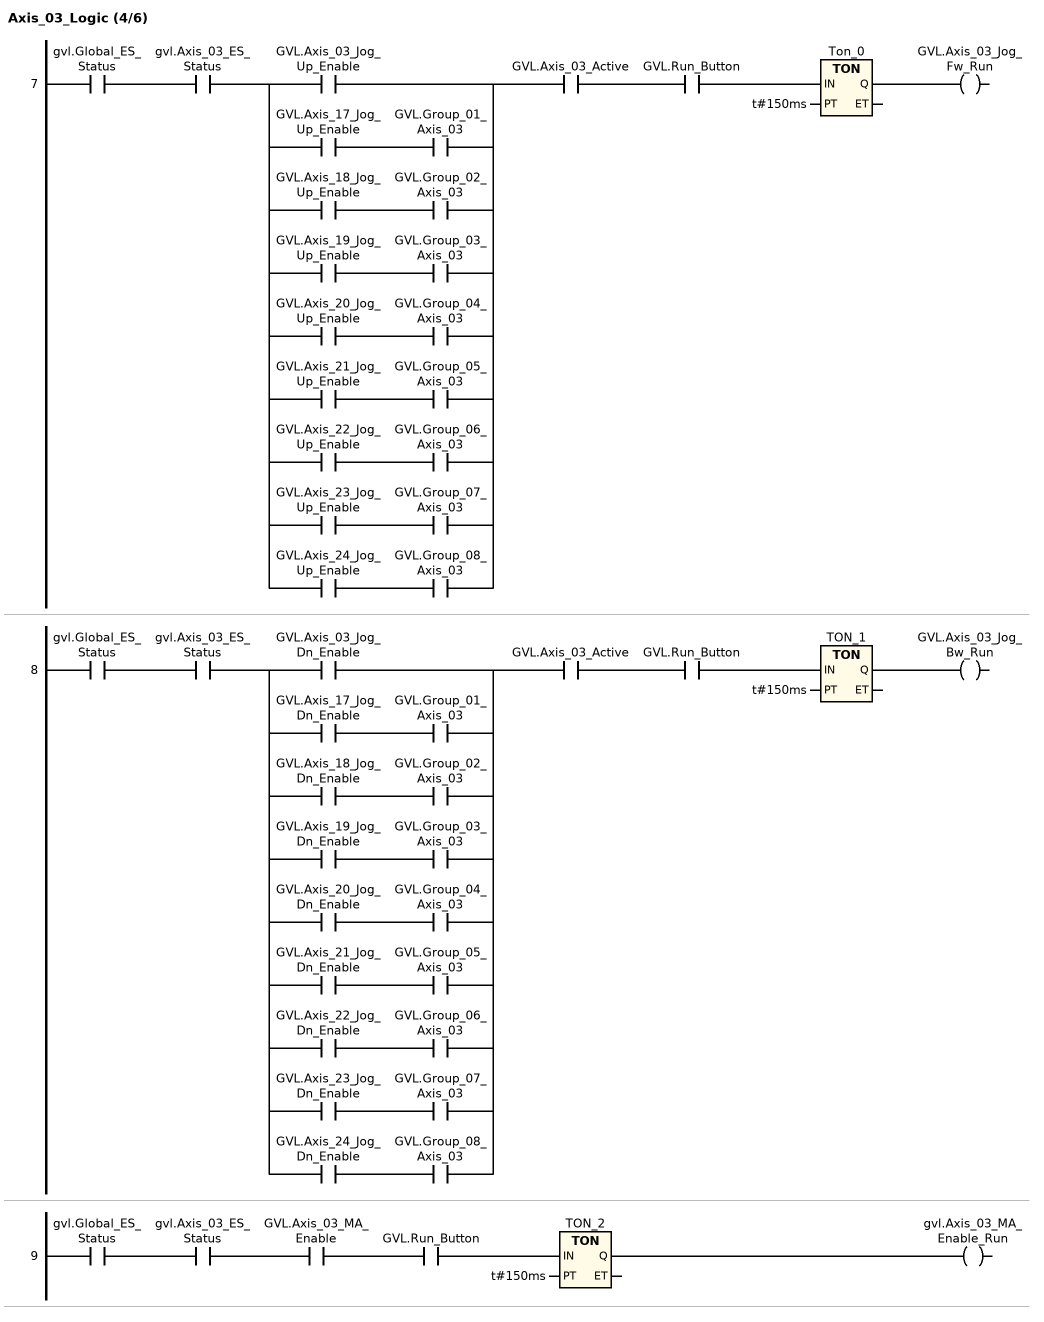
// NETWORK 7
Ton_0(IN := gvl.Global_ES_Status AND gvl.Axis_03_ES_Status AND (GVL.Axis_03_Jog_Up_Enable OR GVL.Axis_17_Jog_Up_Enable AND GVL.Group_01_Axis_03 OR GVL.Axis_18_Jog_Up_Enable AND GVL.Group_02_Axis_03 OR GVL.Axis_19_Jog_Up_Enable AND GVL.Group_03_Axis_03 OR GVL.Axis_20_Jog_Up_Enable AND GVL.Group_04_Axis_03 OR GVL.Axis_21_Jog_Up_Enable AND GVL.Group_05_Axis_03 OR GVL.Axis_22_Jog_Up_Enable AND GVL.Group_06_Axis_03 OR GVL.Axis_23_Jog_Up_Enable AND GVL.Group_07_Axis_03 OR GVL.Axis_24_Jog_Up_Enable AND GVL.Group_08_Axis_03) AND GVL.Axis_03_Active AND GVL.Run_Button, PT := t#150ms); // TON
GVL.Axis_03_Jog_Fw_Run := Ton_0.Q;

// NETWORK 8
TON_1(IN := gvl.Global_ES_Status AND gvl.Axis_03_ES_Status AND (GVL.Axis_03_Jog_Dn_Enable OR GVL.Axis_17_Jog_Dn_Enable AND GVL.Group_01_Axis_03 OR GVL.Axis_18_Jog_Dn_Enable AND GVL.Group_02_Axis_03 OR GVL.Axis_19_Jog_Dn_Enable AND GVL.Group_03_Axis_03 OR GVL.Axis_20_Jog_Dn_Enable AND GVL.Group_04_Axis_03 OR GVL.Axis_21_Jog_Dn_Enable AND GVL.Group_05_Axis_03 OR GVL.Axis_22_Jog_Dn_Enable AND GVL.Group_06_Axis_03 OR GVL.Axis_23_Jog_Dn_Enable AND GVL.Group_07_Axis_03 OR GVL.Axis_24_Jog_Dn_Enable AND GVL.Group_08_Axis_03) AND GVL.Axis_03_Active AND GVL.Run_Button, PT := t#150ms); // TON
GVL.Axis_03_Jog_Bw_Run := TON_1.Q;

// NETWORK 9
TON_2(IN := gvl.Global_ES_Status AND gvl.Axis_03_ES_Status AND GVL.Axis_03_MA_Enable AND GVL.Run_Button, PT := t#150ms); // TON
gvl.Axis_03_MA_Enable_Run := TON_2.Q;

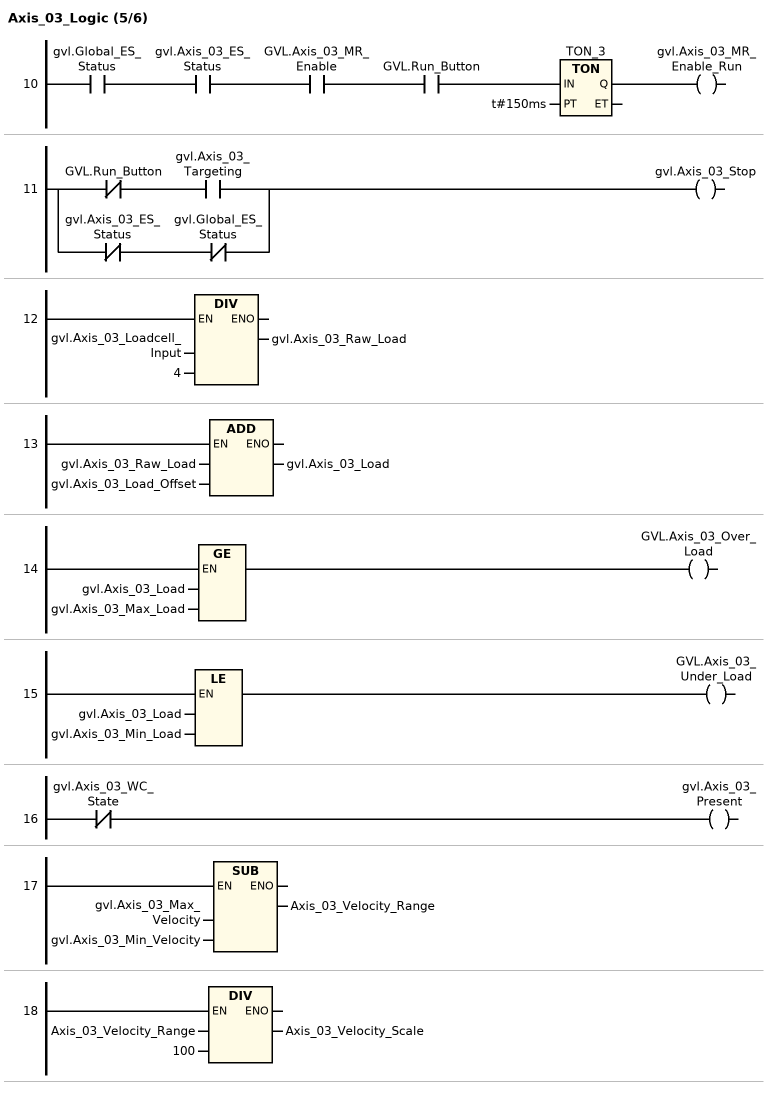
// NETWORK 10
TON_3(IN := gvl.Global_ES_Status AND gvl.Axis_03_ES_Status AND GVL.Axis_03_MR_Enable AND GVL.Run_Button, PT := t#150ms); // TON
gvl.Axis_03_MR_Enable_Run := TON_3.Q;

// NETWORK 11
gvl.Axis_03_Stop := NOT GVL.Run_Button AND gvl.Axis_03_Targeting OR NOT gvl.Axis_03_ES_Status AND NOT gvl.Global_ES_Status;

// NETWORK 12
gvl.Axis_03_Raw_Load := gvl.Axis_03_Loadcell_Input / 4;

// NETWORK 13
gvl.Axis_03_Load := gvl.Axis_03_Raw_Load + gvl.Axis_03_Load_Offset;

// NETWORK 14
GVL.Axis_03_Over_Load := gvl.Axis_03_Load >= gvl.Axis_03_Max_Load;

// NETWORK 15
GVL.Axis_03_Under_Load := gvl.Axis_03_Load <= gvl.Axis_03_Min_Load;

// NETWORK 16
gvl.Axis_03_Present := NOT gvl.Axis_03_WC_State;

// NETWORK 17
Axis_03_Velocity_Range := gvl.Axis_03_Max_Velocity - gvl.Axis_03_Min_Velocity;

// NETWORK 18
Axis_03_Velocity_Scale := Axis_03_Velocity_Range / 100;

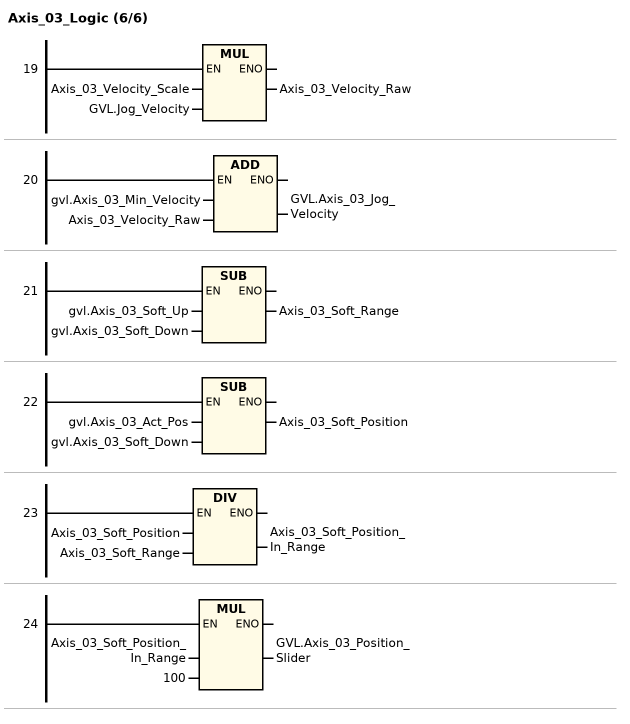
// NETWORK 19
Axis_03_Velocity_Raw := Axis_03_Velocity_Scale * GVL.Jog_Velocity;

// NETWORK 20
GVL.Axis_03_Jog_Velocity := gvl.Axis_03_Min_Velocity + Axis_03_Velocity_Raw;

// NETWORK 21
Axis_03_Soft_Range := gvl.Axis_03_Soft_Up - gvl.Axis_03_Soft_Down;

// NETWORK 22
Axis_03_Soft_Position := gvl.Axis_03_Act_Pos - gvl.Axis_03_Soft_Down;

// NETWORK 23
Axis_03_Soft_Position_In_Range := Axis_03_Soft_Position / Axis_03_Soft_Range;

// NETWORK 24
GVL.Axis_03_Position_Slider := Axis_03_Soft_Position_In_Range * 100;

END_PROGRAM

// ---- POUs/Axis_04_Function_Blocks.TcPOU
PROGRAM Axis_04_Function_Blocks
VAR
END_VAR

